  MoveL 4600 to (-46.03, -30.75, -4) mm, rotated rx 180 ry 0 rz 90 deg; joints [72.359, -18.311, 87.085, 0, 21.226, 72.359]
  Establecer velocidad (1000.0 mm/s)
  MoveL 4601 to (-46.03, -30.75, 10) mm, rotated rx -180 ry 0 rz 90 deg; joints [72.359, -19.035, 87.552, 0, 21.483, 72.359]
  Establecer velocidad (66.7 mm/s)
  MoveL 4602 to (16.92, -66.15, 10) mm, rotated rx -180 ry 0 rz 90 deg; joints [71.876, -17.66, 82.327, 0, 25.333, 71.876]
  MoveL 4603 to (16.92, -66.15, -3.75) mm, rotated rx 180 ry 0 rz 90 deg; joints [71.876, -16.964, 81.867, 0, 25.097, 71.876]
  MoveL 4604 to (16.76, -67.66, -4.16) mm, rotated rx 180 ry 0 rz 90 deg; joints [71.827, -16.937, 81.829, 0, 25.108, 71.827]
  MoveL 4605 to (16.96, -69.17, -4.56) mm, rotated rx -180 ry 0 rz 90 deg; joints [71.782, -16.903, 81.765, 0, 25.138, 71.782]
  MoveL 4606 to (17.5, -70.59, -4.97) mm, rotated rx 180 ry 0 rz 90 deg; joints [71.743, -16.862, 81.678, 0, 25.184, 71.743]
  MoveL 4607 to (18.34, -71.86, -5.37) mm, rotated rx -180 ry 0 rz 90 deg; joints [71.712, -16.816, 81.574, 0, 25.243, 71.712]
  MoveL 4608 to (19.43, -72.91, -5.78) mm, rotated rx -180 ry 0 rz 90 deg; joints [71.69, -16.767, 81.455, 0, 25.311, 71.69]
  MoveL 4609 to (20.74, -73.69, -6.19) mm, rotated rx 180 ry 0 rz 90 deg; joints [71.679, -16.714, 81.328, 0, 25.386, 71.679]
  MoveL 4610 to (22.18, -74.17, -6.59) mm, rotated rx 180 ry 0 rz 90 deg; joints [71.679, -16.662, 81.198, 0, 25.463, 71.679]
  MoveL 4611 to (23.69, -74.28, -7) mm, rotated rx 180 ry 0 rz 90 deg; joints [71.691, -16.609, 81.071, 0, 25.538, 71.691]
  MoveC 4612 to (36.25, -74.06, -7) mm, rotated rx 180 ry 0 rz 90 deg; joints [71.827, -16.352, 80.159, 0, 26.193, 71.827] to (48.8, -73.79, -7) mm, rotated rx -180 ry 0 rz 90 deg; joints [71.962, -16.087, 79.237, 0, 26.85, 71.962]
  MoveC 4613 to (51.44, -70.72, -7) mm, rotated rx -180 ry 0 rz 90 deg; joints [72.082, -16.052, 79.115, 0, 26.937, 72.082] to (51.58, -66.68, -7) mm, rotated rx 180 ry 0 rz 90 deg; joints [72.208, -16.077, 79.201, 0, 26.876, 72.208]
  MoveC 4614 to (38.79, -51.64, -7) mm, rotated rx 180 ry 0 rz 90 deg; joints [72.548, -16.449, 80.502, 0, 25.948, 72.548] to (25.93, -36.65, -7) mm, rotated rx -180 ry 0 rz 90 deg; joints [72.893, -16.807, 81.782, 0, 25.025, 72.893]
  MoveC 4615 to (25.5, -36.2, -7) mm, rotated rx 180 ry 0 rz 90 deg; joints [72.903, -16.818, 81.823, 0, 24.995, 72.903] to (25.04, -35.79, -7) mm, rotated rx -180 ry 0 rz 90 deg; joints [72.911, -16.83, 81.866, 0, 24.964, 72.911]
  MoveL 4616 to (12.33, -25.61, -7) mm, rotated rx 180 ry 0 rz 90 deg; joints [73.111, -17.14, 83.008, 0, 24.132, 73.111]
  MoveL 4617 to (11.85, -25.24, -7) mm, rotated rx -180 ry 0 rz 90 deg; joints [73.118, -17.151, 83.05, 0, 24.101, 73.118]
  MoveC 4618 to (9.1, -24.89, -7) mm, rotated rx 180 ry 0 rz 90 deg; joints [73.102, -17.206, 83.255, 0, 23.951, 73.102] to (6.64, -26.18, -7) mm, rotated rx -180 ry 0 rz 90 deg; joints [73.037, -17.245, 83.402, 0, 23.843, 73.037]
  MoveC 4619 to (6.25, -26.7, -7) mm, rotated rx 180 ry 0 rz 90 deg; joints [73.017, -17.25, 83.419, 0, 23.831, 73.017] to (6, -27.31, -7) mm, rotated rx 180 ry 0 rz 90 deg; joints [72.995, -17.251, 83.424, 0, 23.827, 72.995]
  MoveL 4620 to (-5.3, -69.65, -7) mm, rotated rx 180 ry 0 rz 90 deg; joints [71.534, -17.208, 83.264, 0, 23.945, 71.534]
  MoveC 4621 to (-4.6, -73.1, -7) mm, rotated rx 180 ry 0 rz 90 deg; joints [71.432, -17.173, 83.132, 0, 24.041, 71.432] to (-1.42, -74.62, -7) mm, rotated rx -180 ry 0 rz 90 deg; joints [71.418, -17.103, 82.87, 0, 24.233, 71.418]
  MoveC 4622 to (11.14, -74.47, -7) mm, rotated rx 180 ry 0 rz 90 deg; joints [71.555, -16.86, 81.975, 0, 24.885, 71.555] to (23.69, -74.28, -7) mm, rotated rx 180 ry 0 rz 90 deg; joints [71.691, -16.609, 81.071, 0, 25.538, 71.691]
  MoveL 4623 to (23.57, -66.73, -7) mm, rotated rx -180 ry 0 rz 90 deg; joints [71.925, -16.662, 81.261, 0, 25.401, 71.925]
  MoveL 4624 to (23.57, -66.73, -4) mm, rotated rx -180 ry 0 rz 90 deg; joints [71.925, -16.814, 81.363, 0, 25.451, 71.925]
  Establecer velocidad (1000.0 mm/s)
  MoveL 4625 to (23.57, -66.73, 10) mm, rotated rx 180 ry 0 rz 90 deg; joints [71.925, -17.521, 81.832, 0, 25.689, 71.925]
  Establecer velocidad (66.7 mm/s)
  MoveL 4626 to (64.23, -31.47, 10) mm, rotated rx -180 ry 0 rz 90 deg; joints [73.417, -16.891, 79.643, 0, 27.248, 73.417]
  MoveL 4627 to (64.23, -31.47, -3.75) mm, rotated rx 180 ry 0 rz 90 deg; joints [73.417, -16.202, 79.18, 0, 27.021, 73.417]
  MoveL 4628 to (65.74, -31.65, -4.16) mm, rotated rx 180 ry 0 rz 90 deg; joints [73.425, -16.147, 79.049, 0, 27.098, 73.425]
  MoveL 4629 to (67.24, -31.47, -4.56) mm, rotated rx -180 ry 0 rz 90 deg; joints [73.445, -16.095, 78.926, 0, 27.169, 73.445]
  MoveL 4630 to (68.68, -30.95, -4.97) mm, rotated rx -180 ry 0 rz 90 deg; joints [73.474, -16.046, 78.816, 0, 27.231, 73.474]
  MoveL 4631 to (69.96, -30.14, -5.37) mm, rotated rx 180 ry 0 rz 90 deg; joints [73.511, -16.003, 78.723, 0, 27.279, 73.511]
  MoveL 4632 to (71.03, -29.06, -5.78) mm, rotated rx 180 ry 0 rz 90 deg; joints [73.554, -15.966, 78.653, 0, 27.313, 73.554]
  MoveL 4633 to (71.83, -27.77, -6.19) mm, rotated rx 180 ry 0 rz 90 deg; joints [73.601, -15.936, 78.607, 0, 27.329, 73.601]
  MoveL 4634 to (72.33, -26.33, -6.59) mm, rotated rx -180 ry 0 rz 90 deg; joints [73.65, -15.914, 78.587, 0, 27.327, 73.65]
  MoveL 4635 to (72.47, -24.83, -7) mm, rotated rx 180 ry 0 rz 90 deg; joints [73.698, -15.9, 78.596, 0, 27.304, 73.698]
  MoveL 4636 to (72.47, -13.16, -7) mm, rotated rx 180 ry 0 rz 90 deg; joints [74.059, -15.975, 78.851, 0, 27.124, 74.059]
  MoveC 4637 to (70.6, -10.5, -7) mm, rotated rx 180 ry 0 rz 90 deg; joints [74.125, -16.033, 79.049, 0, 26.983, 74.125] to (67.76, -8.91, -7) mm, rotated rx 180 ry 0 rz 90 deg; joints [74.15, -16.105, 79.297, 0, 26.807, 74.15]
  MoveC 4638 to (66.52, -8.73, -7) mm, rotated rx 180 ry 0 rz 90 deg; joints [74.144, -16.133, 79.394, 0, 26.739, 74.144] to (65.29, -8.93, -7) mm, rotated rx 180 ry 0 rz 90 deg; joints [74.127, -16.158, 79.482, 0, 26.676, 74.127]
  MoveL 4639 to (65.23, -9, -7) mm, rotated rx 180 ry 0 rz 90 deg; joints [74.124, -16.159, 79.485, 0, 26.674, 74.124]
  MoveL 4640 to (54.8, -23.22, -7) mm, rotated rx 180 ry 0 rz 90 deg; joints [73.587, -16.295, 79.957, 0, 26.337, 73.587]
  MoveL 4641 to (54.33, -23.9, -7) mm, rotated rx -180 ry 0 rz 90 deg; joints [73.561, -16.3, 79.977, 0, 26.323, 73.561]
  MoveC 4642 to (53.72, -26.08, -7) mm, rotated rx -180 ry 0 rz 90 deg; joints [73.487, -16.299, 79.974, 0, 26.325, 73.487] to (54.54, -28.19, -7) mm, rotated rx -180 ry 0 rz 90 deg; joints [73.429, -16.269, 79.867, 0, 26.402, 73.429]
  MoveL 4643 to (55.12, -28.9, -7) mm, rotated rx 180 ry 0 rz 90 deg; joints [73.412, -16.252, 79.808, 0, 26.444, 73.412]
  MoveL 4644 to (65.68, -40.76, -7) mm, rotated rx 180 ry 0 rz 90 deg; joints [73.143, -15.946, 78.75, 0, 27.195, 73.143]
  MoveC 4645 to (68.07, -40.73, -7) mm, rotated rx 180 ry 0 rz 90 deg; joints [73.166, -15.893, 78.571, 0, 27.322, 73.166] to (70.2, -39.65, -7) mm, rotated rx 180 ry 0 rz 90 deg; joints [73.22, -15.853, 78.435, 0, 27.418, 73.22]
  MoveL 4646 to (70.46, -39.44, -7) mm, rotated rx 180 ry 0 rz 90 deg; joints [73.228, -15.849, 78.42, 0, 27.429, 73.228]
  MoveC 4647 to (71.67, -38.1, -7) mm, rotated rx -180 ry 0 rz 90 deg; joints [73.281, -15.831, 78.359, 0, 27.472, 73.281] to (72.47, -36.48, -7) mm, rotated rx -180 ry 0 rz 90 deg; joints [73.338, -15.824, 78.335, 0, 27.489, 73.338]
  MoveL 4648 to (72.47, -24.83, -7) mm, rotated rx 180 ry 0 rz 90 deg; joints [73.698, -15.9, 78.596, 0, 27.304, 73.698]
  MoveL 4649 to (64.92, -24.83, -7) mm, rotated rx -180 ry 0 rz 90 deg; joints [73.629, -16.066, 79.165, 0, 26.901, 73.629]
  MoveL 4650 to (64.92, -24.83, -4) mm, rotated rx 180 ry 0 rz 90 deg; joints [73.629, -16.217, 79.268, 0, 26.949, 73.629]
  Establecer velocidad (1000.0 mm/s)
  MoveL 4651 to (64.92, -24.83, 10) mm, rotated rx 180 ry 0 rz 90 deg; joints [73.629, -16.919, 79.739, 0, 27.18, 73.629]
  Establecer velocidad (66.7 mm/s)
  MoveL 4652 to (36.79, 21.66, 10) mm, rotated rx -180 ry 0 rz 90 deg; joints [74.843, -17.788, 82.79, 0, 24.998, 74.843]
  MoveL 4653 to (36.79, 21.66, -3.75) mm, rotated rx -180 ry 0 rz 90 deg; joints [74.843, -17.092, 82.33, 0, 24.762, 74.843]
  MoveL 4654 to (36.94, 23.17, -4.16) mm, rotated rx -180 ry 0 rz 90 deg; joints [74.892, -17.076, 82.335, 0, 24.741, 74.892]
  MoveL 4655 to (36.73, 24.67, -4.56) mm, rotated rx -180 ry 0 rz 90 deg; joints [74.939, -17.068, 82.366, 0, 24.702, 74.939]
  MoveL 4656 to (36.19, 26.09, -4.97) mm, rotated rx 180 ry 0 rz 90 deg; joints [74.979, -17.066, 82.42, 0, 24.646, 74.979]
  MoveL 4657 to (35.35, 27.36, -5.37) mm, rotated rx 180 ry 0 rz 90 deg; joints [75.013, -17.068, 82.492, 0, 24.576, 75.013]
  MoveL 4658 to (34.25, 28.4, -5.78) mm, rotated rx 180 ry 0 rz 90 deg; joints [75.037, -17.075, 82.579, 0, 24.496, 75.037]
  MoveL 4659 to (32.94, 29.18, -6.19) mm, rotated rx 180 ry 0 rz 90 deg; joints [75.05, -17.084, 82.675, 0, 24.409, 75.05]
  MoveL 4660 to (31.49, 29.65, -6.59) mm, rotated rx -180 ry 0 rz 90 deg; joints [75.053, -17.094, 82.776, 0, 24.319, 75.053]
  MoveL 4661 to (29.98, 29.76, -7) mm, rotated rx 180 ry 0 rz 90 deg; joints [75.043, -17.104, 82.874, 0, 24.23, 75.043]
  MoveL 4662 to (10.9, 29.36, -7) mm, rotated rx -180 ry 0 rz 90 deg; joints [74.865, -17.466, 84.239, 0, 23.226, 74.865]
  MoveL 4663 to (9.95, 29.33, -7) mm, rotated rx 180 ry 0 rz 90 deg; joints [74.856, -17.483, 84.306, 0, 23.177, 74.856]
  MoveC 4664 to (7.63, 28.6, -7) mm, rotated rx 180 ry 0 rz 90 deg; joints [74.812, -17.522, 84.457, 0, 23.065, 74.812] to (6.16, 26.68, -7) mm, rotated rx 180 ry 0 rz 90 deg; joints [74.736, -17.54, 84.525, 0, 23.015, 74.736]
  MoveC 4665 to (5.85, 25.43, -7) mm, rotated rx -180 ry 0 rz 90 deg; joints [74.693, -17.539, 84.523, 0, 23.016, 74.693] to (6.04, 24.17, -7) mm, rotated rx 180 ry 0 rz 90 deg; joints [74.653, -17.529, 84.485, 0, 23.045, 74.653]
  MoveL 4666 to (11.41, 9.41, -7) mm, rotated rx -180 ry 0 rz 90 deg; joints [74.225, -17.353, 83.809, 0, 23.544, 74.225]
  MoveC 4667 to (11.94, 8.41, -7) mm, rotated rx -180 ry 0 rz 90 deg; joints [74.197, -17.337, 83.75, 0, 23.587, 74.197] to (12.74, 7.59, -7) mm, rotated rx -180 ry 0 rz 90 deg; joints [74.178, -17.318, 83.676, 0, 23.642, 74.178]
  MoveL 4668 to (28.26, -4.36, -7) mm, rotated rx -180 ry 0 rz 90 deg; joints [73.937, -16.952, 82.311, 0, 24.64, 73.937]
  MoveC 4669 to (29.93, -5.1, -7) mm, rotated rx -180 ry 0 rz 90 deg; joints [73.929, -16.914, 82.175, 0, 24.74, 73.929] to (31.75, -4.99, -7) mm, rotated rx 180 ry 0 rz 90 deg; joints [73.949, -16.879, 82.045, 0, 24.834, 73.949]
  MoveC 4670 to (33.02, -4.44, -7) mm, rotated rx 180 ry 0 rz 90 deg; joints [73.978, -16.857, 81.963, 0, 24.893, 73.978] to (34.03, -3.48, -7) mm, rotated rx -180 ry 0 rz 90 deg; joints [74.018, -16.842, 81.91, 0, 24.932, 74.018]
  MoveL 4671 to (34.59, -2.74, -7) mm, rotated rx 180 ry 0 rz 90 deg; joints [74.047, -16.835, 81.885, 0, 24.95, 74.047]
  MoveL 4672 to (52.72, 22.78, -7) mm, rotated rx -180 ry 0 rz 90 deg; joints [75.015, -16.609, 81.071, 0, 25.538, 75.015]
  MoveC 4673 to (53.21, 23.87, -7) mm, rotated rx 180 ry 0 rz 90 deg; joints [75.054, -16.605, 81.056, 0, 25.549, 75.054] to (53.26, 25.07, -7) mm, rotated rx 180 ry 0 rz 90 deg; joints [75.092, -16.611, 81.076, 0, 25.534, 75.092]
  MoveL 4674 to (53.13, 25.86, -7) mm, rotated rx 180 ry 0 rz 90 deg; joints [75.116, -16.618, 81.101, 0, 25.516, 75.116]
  MoveC 4675 to (52.1, 28.37, -7) mm, rotated rx 180 ry 0 rz 90 deg; joints [75.187, -16.653, 81.227, 0, 25.426, 75.187] to (50.02, 30.11, -7) mm, rotated rx -180 ry 0 rz 90 deg; joints [75.225, -16.705, 81.415, 0, 25.29, 75.225]
  MoveL 4676 to (45.96, 30.09, -7) mm, rotated rx -180 ry 0 rz 90 deg; joints [75.19, -16.788, 81.713, 0, 25.075, 75.19]
  MoveL 4677 to (29.98, 29.76, -7) mm, rotated rx 180 ry 0 rz 90 deg; joints [75.043, -17.104, 82.874, 0, 24.23, 75.043]
  MoveL 4678 to (30.14, 22.21, -7) mm, rotated rx 180 ry 0 rz 90 deg; joints [74.803, -17.061, 82.715, 0, 24.346, 74.803]
  MoveL 4679 to (30.14, 22.21, -4) mm, rotated rx 180 ry 0 rz 90 deg; joints [74.803, -17.214, 82.816, 0, 24.397, 74.803]
  Establecer velocidad (1000.0 mm/s)
  MoveL 4680 to (30.14, 22.21, 10) mm, rotated rx 180 ry 0 rz 90 deg; joints [74.803, -17.924, 83.285, 0, 24.64, 74.803]
  Establecer velocidad (66.7 mm/s)
  MoveL 4681 to (27.33, 65.77, 10) mm, rotated rx -180 ry 0 rz 90 deg; joints [76.185, -18.2, 84.303, 0, 23.897, 76.185]
  MoveL 4682 to (27.33, 65.77, -3.75) mm, rotated rx -180 ry 0 rz 90 deg; joints [76.185, -17.499, 83.844, 0, 23.655, 76.185]
  MoveL 4683 to (27.54, 67.27, -4.16) mm, rotated rx 180 ry 0 rz 90 deg; joints [76.236, -17.481, 83.842, 0, 23.64, 76.236]
  MoveL 4684 to (27.39, 68.78, -4.56) mm, rotated rx 180 ry 0 rz 90 deg; joints [76.284, -17.471, 83.866, 0, 23.605, 76.284]
  MoveL 4685 to (26.9, 70.22, -4.97) mm, rotated rx -180 ry 0 rz 90 deg; joints [76.327, -17.466, 83.913, 0, 23.553, 76.327]
  MoveL 4686 to (26.11, 71.51, -5.37) mm, rotated rx 180 ry 0 rz 90 deg; joints [76.363, -17.466, 83.979, 0, 23.487, 76.363]
  MoveL 4687 to (25.04, 72.6, -5.78) mm, rotated rx 180 ry 0 rz 90 deg; joints [76.39, -17.47, 84.061, 0, 23.41, 76.39]
  MoveL 4688 to (23.77, 73.43, -6.19) mm, rotated rx 180 ry 0 rz 90 deg; joints [76.407, -17.477, 84.153, 0, 23.324, 76.407]
  MoveL 4689 to (22.34, 73.95, -6.59) mm, rotated rx 180 ry 0 rz 90 deg; joints [76.413, -17.486, 84.251, 0, 23.235, 76.413]
  MoveL 4690 to (20.84, 74.12, -7) mm, rotated rx 180 ry 0 rz 90 deg; joints [76.406, -17.494, 84.348, 0, 23.146, 76.406]
  MoveL 4691 to (12.79, 74.25, -7) mm, rotated rx 180 ry 0 rz 90 deg; joints [76.347, -17.643, 84.926, 0, 22.717, 76.347]
  MoveL 4692 to (-26.06, 74.73, -7) mm, rotated rx 180 ry 0 rz 90 deg; joints [76.046, -18.319, 87.663, 0, 20.656, 76.046]
  MoveL 4693 to (-27.17, 74.74, -7) mm, rotated rx -180 ry 0 rz 90 deg; joints [76.037, -18.338, 87.74, 0, 20.597, 76.037]
  MoveC 4694 to (-29.75, 71.47, -7) mm, rotated rx 180 ry 0 rz 90 deg; joints [75.905, -18.366, 87.862, 0, 20.504, 75.905] to (-29.32, 67.32, -7) mm, rotated rx 180 ry 0 rz 90 deg; joints [75.77, -18.342, 87.76, 0, 20.582, 75.77]
  MoveL 4695 to (-10.07, 55.09, -7) mm, rotated rx 180 ry 0 rz 90 deg; joints [75.526, -17.965, 86.203, 0, 21.762, 75.526]
  MoveC 4696 to (-8.73, 54.52, -7) mm, rotated rx 180 ry 0 rz 90 deg; joints [75.519, -17.939, 86.099, 0, 21.84, 75.519] to (-7.29, 54.39, -7) mm, rotated rx 180 ry 0 rz 90 deg; joints [75.527, -17.913, 85.996, 0, 21.918, 75.527]
  MoveL 4697 to (-6.16, 54.47, -7) mm, rotated rx -180 ry 0 rz 90 deg; joints [75.539, -17.894, 85.918, 0, 21.976, 75.539]
  MoveL 4698 to (27.01, 56.93, -7) mm, rotated rx 180 ry 0 rz 90 deg; joints [75.896, -17.297, 83.599, 0, 23.699, 75.896]
  MoveL 4699 to (33.64, 57.46, -7) mm, rotated rx -180 ry 0 rz 90 deg; joints [75.967, -17.172, 83.128, 0, 24.044, 75.967]
  MoveC 4700 to (51.29, 59.11, -7) mm, rotated rx -180 ry 0 rz 90 deg; joints [76.161, -16.83, 81.867, 0, 24.963, 76.161] to (68.87, 61.29, -7) mm, rotated rx 180 ry 0 rz 90 deg; joints [76.367, -16.477, 80.6, 0, 25.877, 76.367]
  MoveC 4701 to (70.75, 62.3, -7) mm, rotated rx 180 ry 0 rz 90 deg; joints [76.414, -16.442, 80.478, 0, 25.965, 76.414] to (71.5, 64.29, -7) mm, rotated rx -180 ry 0 rz 90 deg; joints [76.483, -16.437, 80.458, 0, 25.979, 76.483]
  MoveL 4702 to (71.51, 68.7, -7) mm, rotated rx 180 ry 0 rz 90 deg; joints [76.623, -16.459, 80.536, 0, 25.923, 76.623]
  MoveL 4703 to (71.5, 69.4, -7) mm, rotated rx 180 ry 0 rz 90 deg; joints [76.645, -16.463, 80.549, 0, 25.914, 76.645]
  MoveC 4704 to (70.71, 71.35, -7) mm, rotated rx 180 ry 0 rz 90 deg; joints [76.702, -16.489, 80.643, 0, 25.846, 76.702] to (68.8, 72.25, -7) mm, rotated rx -180 ry 0 rz 90 deg; joints [76.716, -16.534, 80.801, 0, 25.732, 76.716]
  MoveC 4705 to (45.55, 73.46, -7) mm, rotated rx 180 ry 0 rz 90 deg; joints [76.577, -17.015, 82.544, 0, 24.471, 76.577] to (22.27, 74.09, -7) mm, rotated rx -180 ry 0 rz 90 deg; joints [76.417, -17.467, 84.245, 0, 23.222, 76.417]
  MoveL 4706 to (20.84, 74.12, -7) mm, rotated rx 180 ry 0 rz 90 deg; joints [76.406, -17.494, 84.348, 0, 23.146, 76.406]
  MoveL 4707 to (20.71, 66.57, -7) mm, rotated rx 180 ry 0 rz 90 deg; joints [76.158, -17.462, 84.225, 0, 23.237, 76.158]
  MoveL 4708 to (20.71, 66.57, -4) mm, rotated rx 180 ry 0 rz 90 deg; joints [76.158, -17.615, 84.327, 0, 23.288, 76.158]
  Establecer velocidad (1000.0 mm/s)
  MoveL 4709 to (20.71, 66.57, 10) mm, rotated rx 180 ry 0 rz 90 deg; joints [76.158, -18.33, 84.794, 0, 23.536, 76.158]
  Establecer velocidad (66.7 mm/s)
  MoveL 4710 to (27.32, 65.52, 10) mm, rotated rx 180 ry 0 rz 90 deg; joints [76.177, -18.199, 84.299, 0, 23.899, 76.177]
  MoveL 4711 to (27.32, 65.52, -4) mm, rotated rx 180 ry 0 rz 90 deg; joints [76.177, -17.485, 83.832, 0, 23.653, 76.177]
  MoveL 4712 to (27.53, 67.02, -4.41) mm, rotated rx 180 ry 0 rz 90 deg; joints [76.228, -17.468, 83.83, 0, 23.638, 76.228]
  MoveL 4713 to (27.38, 68.53, -4.81) mm, rotated rx -180 ry 0 rz 90 deg; joints [76.276, -17.457, 83.854, 0, 23.603, 76.276]
  MoveL 4714 to (26.89, 69.97, -5.22) mm, rotated rx 180 ry 0 rz 90 deg; joints [76.319, -17.452, 83.9, 0, 23.552, 76.319]
  MoveL 4715 to (26.1, 71.27, -5.63) mm, rotated rx 180 ry 0 rz 90 deg; joints [76.355, -17.452, 83.966, 0, 23.486, 76.355]
  MoveL 4716 to (25.04, 72.36, -6.03) mm, rotated rx -180 ry 0 rz 90 deg; joints [76.382, -17.457, 84.048, 0, 23.408, 76.382]
  MoveL 4717 to (23.76, 73.19, -6.44) mm, rotated rx 180 ry 0 rz 90 deg; joints [76.399, -17.464, 84.141, 0, 23.323, 76.399]
  MoveL 4718 to (22.34, 73.71, -6.84) mm, rotated rx 180 ry 0 rz 90 deg; joints [76.405, -17.472, 84.239, 0, 23.234, 76.405]
  MoveL 4719 to (20.83, 73.88, -7.25) mm, rotated rx -180 ry 0 rz 90 deg; joints [76.398, -17.48, 84.336, 0, 23.144, 76.398]
  MoveC 4720 to (-2.85, 74.25, -7.25) mm, rotated rx 180 ry 0 rz 90 deg; joints [76.221, -17.91, 86.027, 0, 21.884, 76.221] to (-26.54, 74.55, -7.25) mm, rotated rx -180 ry 0 rz 90 deg; joints [76.035, -18.314, 87.685, 0, 20.629, 76.035]
  MoveC 4721 to (-29.11, 71.31, -7.25) mm, rotated rx -180 ry 0 rz 90 deg; joints [75.905, -18.342, 87.806, 0, 20.536, 75.905] to (-28.68, 67.2, -7.25) mm, rotated rx -180 ry 0 rz 90 deg; joints [75.771, -18.318, 87.706, 0, 20.613, 75.771]
  MoveL 4722 to (-27.01, 66.12, -7.25) mm, rotated rx -180 ry 0 rz 90 deg; joints [75.749, -18.286, 87.571, 0, 20.716, 75.749]
  MoveL 4723 to (-11.7, 56.39, -7.25) mm, rotated rx 180 ry 0 rz 90 deg; joints [75.555, -17.986, 86.332, 0, 21.654, 75.555]
  MoveL 4724 to (-9.95, 55.27, -7.25) mm, rotated rx -180 ry 0 rz 90 deg; joints [75.533, -17.951, 86.19, 0, 21.761, 75.533]
  MoveC 4725 to (-8.59, 54.68, -7.25) mm, rotated rx 180 ry 0 rz 90 deg; joints [75.526, -17.925, 86.084, 0, 21.841, 75.526] to (-7.11, 54.59, -7.25) mm, rotated rx 180 ry 0 rz 90 deg; joints [75.535, -17.898, 85.978, 0, 21.92, 75.535]
  MoveL 4726 to (-6.16, 54.66, -7.25) mm, rotated rx 180 ry 0 rz 90 deg; joints [75.545, -17.882, 85.913, 0, 21.969, 75.545]
  MoveL 4727 to (25.11, 56.98, -7.25) mm, rotated rx 180 ry 0 rz 90 deg; joints [75.882, -17.321, 83.728, 0, 23.593, 75.882]
  MoveL 4728 to (32.69, 57.59, -7.25) mm, rotated rx 180 ry 0 rz 90 deg; joints [75.964, -17.178, 83.191, 0, 23.988, 75.964]
  MoveC 4729 to (50.72, 59.32, -7.25) mm, rotated rx 180 ry 0 rz 90 deg; joints [76.163, -16.83, 81.904, 0, 24.926, 76.163] to (68.69, 61.63, -7.25) mm, rotated rx 180 ry 0 rz 90 deg; joints [76.377, -16.47, 80.611, 0, 25.859, 76.377]
  MoveC 4730 to (70.41, 62.54, -7.25) mm, rotated rx 180 ry 0 rz 90 deg; joints [76.419, -16.438, 80.499, 0, 25.939, 76.419] to (71.16, 64.33, -7.25) mm, rotated rx 180 ry 0 rz 90 deg; joints [76.482, -16.432, 80.475, 0, 25.957, 76.482]
  MoveC 4731 to (71.23, 66.85, -7.25) mm, rotated rx -180 ry 0 rz 90 deg; joints [76.562, -16.443, 80.515, 0, 25.928, 76.562] to (71.16, 69.37, -7.25) mm, rotated rx -180 ry 0 rz 90 deg; joints [76.642, -16.457, 80.566, 0, 25.891, 76.642]
  MoveC 4732 to (70.37, 71.13, -7.25) mm, rotated rx -180 ry 0 rz 90 deg; joints [76.692, -16.483, 80.656, 0, 25.827, 76.692] to (68.62, 71.93, -7.25) mm, rotated rx 180 ry 0 rz 90 deg; joints [76.704, -16.523, 80.801, 0, 25.723, 76.704]
  MoveC 4733 to (46.88, 73.13, -7.25) mm, rotated rx 180 ry 0 rz 90 deg; joints [76.577, -16.974, 82.432, 0, 24.542, 76.577] to (25.11, 73.8, -7.25) mm, rotated rx 180 ry 0 rz 90 deg; joints [76.429, -17.4, 84.027, 0, 23.373, 76.429]
  MoveC 4734 to (22.97, 73.84, -7.25) mm, rotated rx -180 ry 0 rz 90 deg; joints [76.414, -17.44, 84.182, 0, 23.258, 76.414] to (20.83, 73.88, -7.25) mm, rotated rx 180 ry 0 rz 90 deg; joints [76.398, -17.48, 84.336, 0, 23.144, 76.398]
  MoveL 4735 to (20.7, 66.33, -7.25) mm, rotated rx -180 ry 0 rz 90 deg; joints [76.15, -17.448, 84.213, 0, 23.235, 76.15]
  MoveL 4736 to (20.7, 66.33, -4.25) mm, rotated rx -180 ry 0 rz 90 deg; joints [76.15, -17.602, 84.315, 0, 23.287, 76.15]
  Establecer velocidad (1000.0 mm/s)
  MoveL 4737 to (20.7, 66.33, 10) mm, rotated rx -180 ry 0 rz 90 deg; joints [76.15, -18.329, 84.791, 0, 23.539, 76.15]
  Establecer velocidad (66.7 mm/s)
  MoveL 4738 to (36.06, 21.39, 10) mm, rotated rx -180 ry 0 rz 90 deg; joints [74.828, -17.802, 82.838, 0, 24.964, 74.828]
  MoveL 4739 to (36.06, 21.39, -4) mm, rotated rx 180 ry 0 rz 90 deg; joints [74.828, -17.092, 82.37, 0, 24.723, 74.828]
  MoveL 4740 to (36.22, 22.9, -4.41) mm, rotated rx -180 ry 0 rz 90 deg; joints [74.878, -17.076, 82.374, 0, 24.702, 74.878]
  MoveL 4741 to (36, 24.41, -4.81) mm, rotated rx -180 ry 0 rz 90 deg; joints [74.924, -17.068, 82.405, 0, 24.663, 74.924]
  MoveL 4742 to (35.46, 25.83, -5.22) mm, rotated rx 180 ry 0 rz 90 deg; joints [74.965, -17.066, 82.459, 0, 24.607, 74.965]
  MoveL 4743 to (34.62, 27.09, -5.63) mm, rotated rx -180 ry 0 rz 90 deg; joints [74.998, -17.069, 82.531, 0, 24.537, 74.998]
  MoveL 4744 to (33.52, 28.14, -6.03) mm, rotated rx 180 ry 0 rz 90 deg; joints [75.022, -17.075, 82.618, 0, 24.457, 75.022]
  MoveL 4745 to (32.22, 28.92, -6.44) mm, rotated rx -180 ry 0 rz 90 deg; joints [75.036, -17.084, 82.714, 0, 24.37, 75.036]
  MoveL 4746 to (30.77, 29.39, -6.84) mm, rotated rx -180 ry 0 rz 90 deg; joints [75.039, -17.095, 82.814, 0, 24.28, 75.039]
  MoveL 4747 to (29.26, 29.5, -7.25) mm, rotated rx -180 ry 0 rz 90 deg; joints [75.029, -17.104, 82.913, 0, 24.191, 75.029]
  MoveL 4748 to (13.74, 29.19, -7.25) mm, rotated rx 180 ry 0 rz 90 deg; joints [74.885, -17.399, 84.024, 0, 23.375, 74.885]
  MoveL 4749 to (9.95, 29.11, -7.25) mm, rotated rx 180 ry 0 rz 90 deg; joints [74.849, -17.469, 84.294, 0, 23.176, 74.849]
  MoveL 4750 to (9, 28.95, -7.25) mm, rotated rx -180 ry 0 rz 90 deg; joints [74.835, -17.486, 84.358, 0, 23.128, 74.835]
  MoveC 4751 to (6.86, 27.27, -7.25) mm, rotated rx -180 ry 0 rz 90 deg; joints [74.762, -17.517, 84.478, 0, 23.039, 74.762] to (6.17, 24.64, -7.25) mm, rotated rx 180 ry 0 rz 90 deg; joints [74.67, -17.517, 84.476, 0, 23.041, 74.67]
  MoveL 4752 to (6.29, 24.17, -7.25) mm, rotated rx -180 ry 0 rz 90 deg; joints [74.656, -17.512, 84.458, 0, 23.054, 74.656]
  MoveL 4753 to (6.64, 23.22, -7.25) mm, rotated rx -180 ry 0 rz 90 deg; joints [74.628, -17.501, 84.415, 0, 23.086, 74.628]
  MoveL 4754 to (11.66, 9.42, -7.25) mm, rotated rx 180 ry 0 rz 90 deg; joints [74.227, -17.335, 83.782, 0, 23.553, 74.227]
  MoveC 4755 to (12.05, 8.66, -7.25) mm, rotated rx 180 ry 0 rz 90 deg; joints [74.206, -17.324, 83.739, 0, 23.585, 74.206] to (12.61, 8.02, -7.25) mm, rotated rx -180 ry 0 rz 90 deg; joints [74.191, -17.31, 83.686, 0, 23.624, 74.191]
  MoveL 4756 to (12.79, 7.85, -7.25) mm, rotated rx -180 ry 0 rz 90 deg; joints [74.187, -17.306, 83.669, 0, 23.636, 74.187]
  MoveL 4757 to (27.96, -3.81, -7.25) mm, rotated rx 180 ry 0 rz 90 deg; joints [73.952, -16.948, 82.337, 0, 24.612, 73.952]
  MoveL 4758 to (28.9, -4.48, -7.25) mm, rotated rx 180 ry 0 rz 90 deg; joints [73.94, -16.926, 82.254, 0, 24.672, 73.94]
  MoveC 4759 to (31.69, -4.67, -7.25) mm, rotated rx -180 ry 0 rz 90 deg; joints [73.959, -16.869, 82.047, 0, 24.822, 73.959] to (34.01, -3.1, -7.25) mm, rotated rx 180 ry 0 rz 90 deg; joints [74.03, -16.832, 81.911, 0, 24.921, 74.03]
  MoveL 4760 to (34.56, -2.37, -7.25) mm, rotated rx -180 ry 0 rz 90 deg; joints [74.058, -16.825, 81.886, 0, 24.939, 74.058]
  MoveL 4761 to (52.59, 23.08, -7.25) mm, rotated rx -180 ry 0 rz 90 deg; joints [75.023, -16.601, 81.078, 0, 25.523, 75.023]
  MoveC 4762 to (52.24, 27, -7.25) mm, rotated rx 180 ry 0 rz 90 deg; joints [75.145, -16.63, 81.181, 0, 25.449, 75.145] to (49.53, 29.85, -7.25) mm, rotated rx -180 ry 0 rz 90 deg; joints [75.212, -16.701, 81.437, 0, 25.264, 75.212]
  MoveL 4763 to (45.96, 29.83, -7.25) mm, rotated rx 180 ry 0 rz 90 deg; joints [75.182, -16.774, 81.7, 0, 25.074, 75.182]
  MoveL 4764 to (29.26, 29.5, -7.25) mm, rotated rx -180 ry 0 rz 90 deg; joints [75.029, -17.104, 82.913, 0, 24.191, 75.029]
  MoveL 4765 to (29.41, 21.95, -7.25) mm, rotated rx 180 ry 0 rz 90 deg; joints [74.788, -17.061, 82.754, 0, 24.307, 74.788]
  MoveL 4766 to (29.41, 21.95, -4.25) mm, rotated rx -180 ry 0 rz 90 deg; joints [74.788, -17.214, 82.856, 0, 24.358, 74.788]
  Establecer velocidad (1000.0 mm/s)
  MoveL 4767 to (29.41, 21.95, 10) mm, rotated rx 180 ry 0 rz 90 deg; joints [74.788, -17.937, 83.332, 0, 24.605, 74.788]
  Establecer velocidad (66.7 mm/s)
  MoveL 4768 to (63.96, -31.55, 10) mm, rotated rx -180 ry 0 rz 90 deg; joints [73.412, -16.896, 79.662, 0, 27.235, 73.412]
  MoveL 4769 to (63.96, -31.55, -4) mm, rotated rx 180 ry 0 rz 90 deg; joints [73.412, -16.195, 79.19, 0, 27.004, 73.412]
  MoveL 4770 to (65.46, -31.73, -4.41) mm, rotated rx -180 ry 0 rz 90 deg; joints [73.42, -16.14, 79.059, 0, 27.081, 73.42]
  MoveL 4771 to (66.97, -31.55, -4.81) mm, rotated rx 180 ry 0 rz 90 deg; joints [73.44, -16.088, 78.936, 0, 27.152, 73.44]
  MoveL 4772 to (68.4, -31.04, -5.22) mm, rotated rx 180 ry 0 rz 90 deg; joints [73.469, -16.039, 78.826, 0, 27.213, 73.469]
  MoveL 4773 to (69.68, -30.22, -5.63) mm, rotated rx 180 ry 0 rz 90 deg; joints [73.506, -15.996, 78.734, 0, 27.262, 73.506]
  MoveL 4774 to (70.76, -29.14, -6.03) mm, rotated rx -180 ry 0 rz 90 deg; joints [73.549, -15.959, 78.663, 0, 27.296, 73.549]
  MoveL 4775 to (71.56, -27.85, -6.44) mm, rotated rx -180 ry 0 rz 90 deg; joints [73.596, -15.929, 78.617, 0, 27.312, 73.596]
  MoveL 4776 to (72.06, -26.42, -6.84) mm, rotated rx 180 ry 0 rz 90 deg; joints [73.645, -15.907, 78.597, 0, 27.31, 73.645]
  MoveL 4777 to (72.2, -24.91, -7.25) mm, rotated rx -180 ry 0 rz 90 deg; joints [73.693, -15.893, 78.606, 0, 27.287, 73.693]
  MoveL 4778 to (72.2, -13.88, -7.25) mm, rotated rx 180 ry 0 rz 90 deg; joints [74.035, -15.964, 78.847, 0, 27.117, 74.035]
  MoveC 4779 to (70.43, -11.3, -7.25) mm, rotated rx -180 ry 0 rz 90 deg; joints [74.099, -16.019, 79.036, 0, 26.983, 74.099] to (67.76, -9.69, -7.25) mm, rotated rx 180 ry 0 rz 90 deg; joints [74.125, -16.087, 79.272, 0, 26.815, 74.125]
  MoveC 4780 to (66.44, -9.46, -7.25) mm, rotated rx 180 ry 0 rz 90 deg; joints [74.121, -16.117, 79.376, 0, 26.741, 74.121] to (65.12, -9.62, -7.25) mm, rotated rx 180 ry 0 rz 90 deg; joints [74.104, -16.145, 79.472, 0, 26.673, 74.104]
  MoveL 4781 to (55.13, -23.22, -7.25) mm, rotated rx 180 ry 0 rz 90 deg; joints [73.59, -16.275, 79.924, 0, 26.351, 73.59]
  MoveL 4782 to (54.65, -23.93, -7.25) mm, rotated rx 180 ry 0 rz 90 deg; joints [73.563, -16.281, 79.944, 0, 26.336, 73.563]
  MoveC 4783 to (54.05, -26.08, -7.25) mm, rotated rx -180 ry 0 rz 90 deg; joints [73.49, -16.28, 79.942, 0, 26.338, 73.49] to (54.86, -28.16, -7.25) mm, rotated rx 180 ry 0 rz 90 deg; joints [73.433, -16.249, 79.835, 0, 26.414, 73.433]
  MoveL 4784 to (55.44, -28.85, -7.25) mm, rotated rx 180 ry 0 rz 90 deg; joints [73.417, -16.233, 79.777, 0, 26.456, 73.417]
  MoveL 4785 to (65.51, -40.15, -7.25) mm, rotated rx 180 ry 0 rz 90 deg; joints [73.16, -15.941, 78.769, 0, 27.172, 73.16]
  MoveC 4786 to (68.03, -40.02, -7.25) mm, rotated rx 180 ry 0 rz 90 deg; joints [73.188, -15.886, 78.582, 0, 27.305, 73.188] to (70.24, -38.8, -7.25) mm, rotated rx 180 ry 0 rz 90 deg; joints [73.246, -15.845, 78.443, 0, 27.403, 73.246]
  MoveC 4787 to (71.39, -37.49, -7.25) mm, rotated rx 180 ry 0 rz 90 deg; joints [73.297, -15.829, 78.385, 0, 27.443, 73.297] to (72.2, -35.94, -7.25) mm, rotated rx 180 ry 0 rz 90 deg; joints [73.352, -15.821, 78.359, 0, 27.462, 73.352]
  MoveL 4788 to (72.2, -24.91, -7.25) mm, rotated rx -180 ry 0 rz 90 deg; joints [73.693, -15.893, 78.606, 0, 27.287, 73.693]
  MoveL 4789 to (64.65, -24.91, -7.25) mm, rotated rx -180 ry 0 rz 90 deg; joints [73.624, -16.059, 79.175, 0, 26.884, 73.624]
  MoveL 4790 to (64.65, -24.91, -4.25) mm, rotated rx 180 ry 0 rz 90 deg; joints [73.624, -16.21, 79.278, 0, 26.932, 73.624]
  Establecer velocidad (1000.0 mm/s)
  MoveL 4791 to (64.65, -24.91, 10) mm, rotated rx 180 ry 0 rz 90 deg; joints [73.624, -16.924, 79.757, 0, 27.167, 73.624]
  Establecer velocidad (66.7 mm/s)
  MoveL 4792 to (16.48, -65.93, 10) mm, rotated rx 180 ry 0 rz 90 deg; joints [71.878, -17.67, 82.364, 0, 25.306, 71.878]
  MoveL 4793 to (16.48, -65.93, -4) mm, rotated rx -180 ry 0 rz 90 deg; joints [71.878, -16.962, 81.895, 0, 25.067, 71.878]
  MoveL 4794 to (16.32, -67.44, -4.41) mm, rotated rx 180 ry 0 rz 90 deg; joints [71.829, -16.935, 81.857, 0, 25.077, 71.829]
  MoveL 4795 to (16.53, -68.94, -4.81) mm, rotated rx 180 ry 0 rz 90 deg; joints [71.784, -16.9, 81.793, 0, 25.107, 71.784]
  MoveL 4796 to (17.06, -70.37, -5.22) mm, rotated rx -180 ry 0 rz 90 deg; joints [71.745, -16.859, 81.707, 0, 25.153, 71.745]
  MoveL 4797 to (17.9, -71.63, -5.63) mm, rotated rx 180 ry 0 rz 90 deg; joints [71.714, -16.814, 81.602, 0, 25.212, 71.714]
  MoveL 4798 to (19, -72.68, -6.03) mm, rotated rx -180 ry 0 rz 90 deg; joints [71.693, -16.764, 81.483, 0, 25.281, 71.693]
  MoveL 4799 to (20.3, -73.47, -6.44) mm, rotated rx 180 ry 0 rz 90 deg; joints [71.682, -16.712, 81.357, 0, 25.356, 71.682]
  MoveL 4800 to (21.75, -73.94, -6.84) mm, rotated rx -180 ry 0 rz 90 deg; joints [71.682, -16.659, 81.226, 0, 25.433, 71.682]
  MoveL 4801 to (23.26, -74.06, -7.25) mm, rotated rx -180 ry 0 rz 90 deg; joints [71.694, -16.607, 81.1, 0, 25.507, 71.694]
  MoveC 4802 to (35.8, -73.82, -7.25) mm, rotated rx -180 ry 0 rz 90 deg; joints [71.83, -16.35, 80.189, 0, 26.161, 71.83] to (48.33, -73.53, -7.25) mm, rotated rx 180 ry 0 rz 90 deg; joints [71.965, -16.087, 79.269, 0, 26.817, 71.965]
  MoveC 4803 to (50.92, -70.47, -7.25) mm, rotated rx -180 ry 0 rz 90 deg; joints [72.085, -16.052, 79.151, 0, 26.902, 72.085] to (51.06, -66.46, -7.25) mm, rotated rx 180 ry 0 rz 90 deg; joints [72.21, -16.077, 79.236, 0, 26.841, 72.21]
  MoveC 4804 to (38.31, -51.44, -7.25) mm, rotated rx 180 ry 0 rz 90 deg; joints [72.55, -16.448, 80.533, 0, 25.915, 72.55] to (25.48, -36.48, -7.25) mm, rotated rx 180 ry 0 rz 90 deg; joints [72.894, -16.804, 81.81, 0, 24.994, 72.894]
  MoveL 4805 to (25.11, -36.14, -7.25) mm, rotated rx 180 ry 0 rz 90 deg; joints [72.901, -16.814, 81.844, 0, 24.969, 72.901]
  MoveL 4806 to (20.82, -32.69, -7.25) mm, rotated rx 180 ry 0 rz 90 deg; joints [72.968, -16.92, 82.232, 0, 24.688, 72.968]
  MoveL 4807 to (19.65, -31.75, -7.25) mm, rotated rx 180 ry 0 rz 90 deg; joints [72.987, -16.948, 82.337, 0, 24.611, 72.987]
  MoveL 4808 to (12.56, -26.06, -7.25) mm, rotated rx -180 ry 0 rz 90 deg; joints [73.099, -17.12, 82.973, 0, 24.148, 73.099]
  MoveL 4809 to (12.22, -25.78, -7.25) mm, rotated rx -180 ry 0 rz 90 deg; joints [73.104, -17.128, 83.003, 0, 24.125, 73.104]
  MoveC 4810 to (9.73, -25.16, -7.25) mm, rotated rx 180 ry 0 rz 90 deg; joints [73.1, -17.18, 83.195, 0, 23.984, 73.1] to (7.32, -26.06, -7.25) mm, rotated rx -180 ry 0 rz 90 deg; joints [73.048, -17.22, 83.348, 0, 23.873, 73.048]
  MoveL 4811 to (7.22, -26.13, -7.25) mm, rotated rx 180 ry 0 rz 90 deg; joints [73.045, -17.222, 83.353, 0, 23.868, 73.045]
  MoveC 4812 to (6.54, -26.82, -7.25) mm, rotated rx 180 ry 0 rz 90 deg; joints [73.016, -17.231, 83.387, 0, 23.844, 73.016] to (6.13, -27.7, -7.25) mm, rotated rx 180 ry 0 rz 90 deg; joints [72.984, -17.233, 83.397, 0, 23.836, 72.984]
  MoveL 4813 to (-5.06, -69.65, -7.25) mm, rotated rx 180 ry 0 rz 90 deg; joints [71.537, -17.191, 83.239, 0, 23.953, 71.537]
  MoveC 4814 to (-5.09, -71.39, -7.25) mm, rotated rx 180 ry 0 rz 90 deg; joints [71.481, -17.181, 83.199, 0, 23.982, 71.481] to (-4.26, -72.93, -7.25) mm, rotated rx -180 ry 0 rz 90 deg; joints [71.441, -17.155, 83.104, 0, 24.051, 71.441]
  MoveC 4815 to (-3.18, -73.89, -7.25) mm, rotated rx -180 ry 0 rz 90 deg; joints [71.423, -17.129, 83.004, 0, 24.125, 71.423] to (-1.82, -74.39, -7.25) mm, rotated rx 180 ry 0 rz 90 deg; joints [71.421, -17.099, 82.895, 0, 24.204, 71.421]
  MoveC 4816 to (10.72, -74.25, -7.25) mm, rotated rx 180 ry 0 rz 90 deg; joints [71.558, -16.857, 82.002, 0, 24.855, 71.558] to (23.26, -74.06, -7.25) mm, rotated rx -180 ry 0 rz 90 deg; joints [71.694, -16.607, 81.1, 0, 25.507, 71.694]
  MoveL 4817 to (23.13, -66.51, -7.25) mm, rotated rx -180 ry 0 rz 90 deg; joints [71.928, -16.66, 81.29, 0, 25.37, 71.928]
  MoveL 4818 to (23.13, -66.51, -4.25) mm, rotated rx -180 ry 0 rz 90 deg; joints [71.928, -16.812, 81.392, 0, 25.42, 71.928]
  Establecer velocidad (1000.0 mm/s)
  MoveL 4819 to (23.13, -66.51, 10) mm, rotated rx 180 ry 0 rz 90 deg; joints [71.928, -17.531, 81.869, 0, 25.662, 71.928]
  Establecer velocidad (66.7 mm/s)
  MoveL 4820 to (-35.06, -51.48, 10) mm, rotated rx 180 ry 0 rz 90 deg; joints [71.8, -18.73, 86.336, 0, 22.394, 71.8]
  MoveL 4821 to (-35.06, -51.48, -4) mm, rotated rx 180 ry 0 rz 90 deg; joints [71.8, -18.011, 85.869, 0, 22.141, 71.8]
  MoveL 4822 to (-33.65, -52.04, -4.41) mm, rotated rx -180 ry 0 rz 90 deg; joints [71.797, -17.962, 85.745, 0, 22.217, 71.797]
  MoveL 4823 to (-32.14, -52.25, -4.81) mm, rotated rx -180 ry 0 rz 90 deg; joints [71.806, -17.914, 85.623, 0, 22.291, 71.806]
  MoveL 4824 to (-30.63, -52.11, -5.22) mm, rotated rx -180 ry 0 rz 90 deg; joints [71.826, -17.867, 85.507, 0, 22.36, 71.826]
  MoveL 4825 to (-29.18, -51.65, -5.63) mm, rotated rx 180 ry 0 rz 90 deg; joints [71.857, -17.824, 85.404, 0, 22.42, 71.857]
  MoveL 4826 to (-27.87, -50.87, -6.03) mm, rotated rx 180 ry 0 rz 90 deg; joints [71.895, -17.784, 85.317, 0, 22.467, 71.895]
  MoveL 4827 to (-26.77, -49.83, -6.44) mm, rotated rx 180 ry 0 rz 90 deg; joints [71.941, -17.75, 85.25, 0, 22.5, 71.941]
  MoveL 4828 to (-25.92, -48.57, -6.84) mm, rotated rx -180 ry 0 rz 90 deg; joints [71.99, -17.721, 85.206, 0, 22.515, 71.99]
  MoveL 4829 to (-25.41, -47.14, -7.25) mm, rotated rx 180 ry 0 rz 90 deg; joints [72.042, -17.7, 85.189, 0, 22.511, 72.042]
  MoveL 4830 to (-19.66, -25.11, -7.25) mm, rotated rx 180 ry 0 rz 90 deg; joints [72.812, -17.721, 85.274, 0, 22.447, 72.812]
  MoveL 4831 to (-19.17, -23.22, -7.25) mm, rotated rx -180 ry 0 rz 90 deg; joints [72.878, -17.723, 85.281, 0, 22.442, 72.878]
  MoveL 4832 to (-19.06, -22.62, -7.25) mm, rotated rx 180 ry 0 rz 90 deg; joints [72.899, -17.724, 85.286, 0, 22.438, 72.899]
  MoveC 4833 to (-19.03, -21.94, -7.25) mm, rotated rx 180 ry 0 rz 90 deg; joints [72.921, -17.727, 85.298, 0, 22.429, 72.921] to (-19.19, -21.27, -7.25) mm, rotated rx -180 ry 0 rz 90 deg; joints [72.941, -17.734, 85.324, 0, 22.41, 72.941]
  MoveL 4834 to (-19.35, -20.88, -7.25) mm, rotated rx 180 ry 0 rz 90 deg; joints [72.952, -17.739, 85.344, 0, 22.395, 72.952]
  MoveC 4835 to (-20.69, -19.13, -7.25) mm, rotated rx -180 ry 0 rz 90 deg; joints [72.996, -17.772, 85.475, 0, 22.297, 72.996] to (-22.74, -18.33, -7.25) mm, rotated rx 180 ry 0 rz 90 deg; joints [73.001, -17.812, 85.635, 0, 22.178, 73.001]
  MoveL 4836 to (-23.22, -18.38, -7.25) mm, rotated rx -180 ry 0 rz 90 deg; joints [72.995, -17.82, 85.667, 0, 22.154, 72.995]
  MoveL 4837 to (-26.06, -18.97, -7.25) mm, rotated rx 180 ry 0 rz 90 deg; joints [72.947, -17.867, 85.852, 0, 22.015, 72.947]
  MoveL 4838 to (-71.94, -28.73, -7.25) mm, rotated rx 180 ry 0 rz 90 deg; joints [72.152, -18.568, 88.773, 0, 19.794, 72.152]
  MoveC 4839 to (-72.61, -28.92, -7.25) mm, rotated rx -180 ry 0 rz 90 deg; joints [72.139, -18.577, 88.814, 0, 19.763, 72.139] to (-73.24, -29.19, -7.25) mm, rotated rx 180 ry 0 rz 90 deg; joints [72.123, -18.585, 88.851, 0, 19.735, 72.123]
  MoveC 4840 to (-74.66, -30.5, -7.25) mm, rotated rx -180 ry 0 rz 90 deg; joints [72.064, -18.6, 88.917, 0, 19.683, 72.064] to (-75.18, -32.35, -7.25) mm, rotated rx 180 ry 0 rz 90 deg; joints [71.997, -18.599, 88.912, 0, 19.688, 71.997]
  MoveL 4841 to (-75.18, -70.81, -7.25) mm, rotated rx -180 ry 0 rz 90 deg; joints [70.728, -18.398, 88.043, 0, 20.355, 70.728]
  MoveC 4842 to (-74.95, -72.13, -7.25) mm, rotated rx -180 ry 0 rz 90 deg; joints [70.688, -18.387, 87.997, 0, 20.39, 70.688] to (-74.28, -73.29, -7.25) mm, rotated rx -180 ry 0 rz 90 deg; joints [70.657, -18.37, 87.925, 0, 20.445, 70.657]
  MoveC 4843 to (-73.04, -74.19, -7.25) mm, rotated rx 180 ry 0 rz 90 deg; joints [70.642, -18.346, 87.821, 0, 20.525, 70.642] to (-71.55, -74.53, -7.25) mm, rotated rx 180 ry 0 rz 90 deg; joints [70.648, -18.32, 87.712, 0, 20.608, 70.648]
  MoveL 4844 to (-70.6, -74.54, -7.25) mm, rotated rx -180 ry 0 rz 90 deg; joints [70.659, -18.305, 87.648, 0, 20.657, 70.659]
  MoveL 4845 to (-35.3, -74.26, -7.25) mm, rotated rx 180 ry 0 rz 90 deg; joints [71.064, -17.714, 85.247, 0, 22.467, 71.064]
  MoveC 4846 to (-33.13, -73.52, -7.25) mm, rotated rx -180 ry 0 rz 90 deg; joints [71.111, -17.681, 85.115, 0, 22.566, 71.111] to (-31.82, -71.64, -7.25) mm, rotated rx -180 ry 0 rz 90 deg; joints [71.186, -17.669, 85.068, 0, 22.601, 71.186]
  MoveL 4847 to (-31.51, -70.6, -7.25) mm, rotated rx 180 ry 0 rz 90 deg; joints [71.223, -17.67, 85.071, 0, 22.598, 71.223]
  MoveL 4848 to (-28.07, -57.33, -7.25) mm, rotated rx -180 ry 0 rz 90 deg; joints [71.686, -17.687, 85.141, 0, 22.546, 71.686]
  MoveL 4849 to (-25.41, -47.14, -7.25) mm, rotated rx 180 ry 0 rz 90 deg; joints [72.042, -17.7, 85.189, 0, 22.511, 72.042]
  MoveL 4850 to (-32.71, -45.23, -7.25) mm, rotated rx 180 ry 0 rz 90 deg; joints [72.027, -17.838, 85.739, 0, 22.1, 72.027]
  MoveL 4851 to (-32.71, -45.23, -4.25) mm, rotated rx 180 ry 0 rz 90 deg; joints [72.027, -17.993, 85.84, 0, 22.153, 72.027]
  Establecer velocidad (1000.0 mm/s)
  MoveL 4852 to (-32.71, -45.23, 10) mm, rotated rx 180 ry 0 rz 90 deg; joints [72.027, -18.725, 86.315, 0, 22.41, 72.027]
  Establecer velocidad (66.7 mm/s)
  MoveL 4853 to (-66.94, 36.36, 10) mm, rotated rx 180 ry 0 rz 90 deg; joints [74.388, -19.691, 90.328, 0, 19.363, 74.388]
  MoveL 4854 to (-66.94, 36.36, -4) mm, rotated rx -180 ry 0 rz 90 deg; joints [74.388, -18.958, 89.861, 0, 19.098, 74.388]
  MoveL 4855 to (-68.44, 36.55, -4.41) mm, rotated rx 180 ry 0 rz 90 deg; joints [74.38, -18.96, 89.952, 0, 19.009, 74.38]
  MoveL 4856 to (-69.95, 36.37, -4.81) mm, rotated rx -180 ry 0 rz 90 deg; joints [74.359, -18.961, 90.036, 0, 18.925, 74.359]
  MoveL 4857 to (-71.38, 35.85, -5.22) mm, rotated rx -180 ry 0 rz 90 deg; joints [74.328, -18.958, 90.108, 0, 18.85, 74.328]
  MoveL 4858 to (-72.66, 35.04, -5.63) mm, rotated rx 180 ry 0 rz 90 deg; joints [74.288, -18.953, 90.165, 0, 18.788, 74.288]
  MoveL 4859 to (-73.73, 33.96, -6.03) mm, rotated rx 180 ry 0 rz 90 deg; joints [74.241, -18.942, 90.202, 0, 18.74, 74.241]
  MoveL 4860 to (-74.54, 32.67, -6.44) mm, rotated rx -180 ry 0 rz 90 deg; joints [74.19, -18.928, 90.218, 0, 18.71, 74.19]
  MoveL 4861 to (-75.04, 31.23, -6.84) mm, rotated rx 180 ry 0 rz 90 deg; joints [74.136, -18.908, 90.21, 0, 18.697, 74.136]
  MoveL 4862 to (-75.18, 29.72, -7.25) mm, rotated rx 180 ry 0 rz 90 deg; joints [74.083, -18.882, 90.177, 0, 18.705, 74.083]
  MoveL 4863 to (-75.18, 1.42, -7.25) mm, rotated rx 180 ry 0 rz 90 deg; joints [73.126, -18.759, 89.621, 0, 19.138, 73.126]
  MoveL 4864 to (-75.16, 0.57, -7.25) mm, rotated rx -180 ry 0 rz 90 deg; joints [73.098, -18.755, 89.602, 0, 19.153, 73.098]
  MoveC 4865 to (-74.13, -1.88, -7.25) mm, rotated rx -180 ry 0 rz 90 deg; joints [73.026, -18.729, 89.484, 0, 19.245, 73.026] to (-71.72, -2.96, -7.25) mm, rotated rx 180 ry 0 rz 90 deg; joints [73.015, -18.687, 89.3, 0, 19.387, 73.015]
  MoveC 4866 to (-71.04, -2.95, -7.25) mm, rotated rx -180 ry 0 rz 90 deg; joints [73.022, -18.677, 89.255, 0, 19.422, 73.022] to (-70.37, -2.84, -7.25) mm, rotated rx -180 ry 0 rz 90 deg; joints [73.032, -18.668, 89.213, 0, 19.455, 73.032]
  MoveC 4867 to (-45.68, 2.82, -7.25) mm, rotated rx 180 ry 0 rz 90 deg; joints [73.469, -18.307, 87.656, 0, 20.65, 73.469] to (-20.99, 8.51, -7.25) mm, rotated rx 180 ry 0 rz 90 deg; joints [73.894, -17.921, 86.068, 0, 21.853, 73.894]
  MoveC 4868 to (-18.56, 10.33, -7.25) mm, rotated rx -180 ry 0 rz 90 deg; joints [73.977, -17.888, 85.936, 0, 21.952, 73.977] to (-18.29, 13.35, -7.25) mm, rotated rx 180 ry 0 rz 90 deg; joints [74.078, -17.898, 85.977, 0, 21.921, 74.078]
  MoveL 4869 to (-18.74, 14.69, -7.25) mm, rotated rx 180 ry 0 rz 90 deg; joints [74.118, -17.912, 86.035, 0, 21.877, 74.118]
  MoveL 4870 to (-24.52, 30.8, -7.25) mm, rotated rx -180 ry 0 rz 90 deg; joints [74.595, -18.089, 86.751, 0, 21.338, 74.595]
  MoveL 4871 to (-25.11, 32.4, -7.25) mm, rotated rx 180 ry 0 rz 90 deg; joints [74.643, -18.106, 86.823, 0, 21.284, 74.643]
  MoveL 4872 to (-25.17, 32.55, -7.25) mm, rotated rx -180 ry 0 rz 90 deg; joints [74.647, -18.108, 86.829, 0, 21.279, 74.647]
  MoveC 4873 to (-25.72, 33.5, -7.25) mm, rotated rx -180 ry 0 rz 90 deg; joints [74.674, -18.122, 86.886, 0, 21.236, 74.674] to (-26.54, 34.24, -7.25) mm, rotated rx 180 ry 0 rz 90 deg; joints [74.691, -18.139, 86.956, 0, 21.182, 74.691]
  MoveL 4874 to (-27.96, 35.18, -7.25) mm, rotated rx -180 ry 0 rz 90 deg; joints [74.709, -18.167, 87.072, 0, 21.095, 74.709]
  MoveL 4875 to (-64.01, 58.28, -7.25) mm, rotated rx 180 ry 0 rz 90 deg; joints [75.16, -18.833, 89.955, 0, 18.879, 75.16]
  MoveL 4876 to (-68.7, 61.3, -7.25) mm, rotated rx -180 ry 0 rz 90 deg; joints [75.221, -18.914, 90.324, 0, 18.59, 75.221]
  MoveC 4877 to (-69.62, 61.83, -7.25) mm, rotated rx -180 ry 0 rz 90 deg; joints [75.23, -18.929, 90.394, 0, 18.535, 75.23] to (-70.6, 62.22, -7.25) mm, rotated rx -180 ry 0 rz 90 deg; joints [75.235, -18.945, 90.467, 0, 18.478, 75.235]
  MoveC 4878 to (-73.29, 61.74, -7.25) mm, rotated rx 180 ry 0 rz 90 deg; joints [75.194, -18.982, 90.638, 0, 18.344, 75.194] to (-75.06, 59.66, -7.25) mm, rotated rx 180 ry 0 rz 90 deg; joints [75.107, -19, 90.72, 0, 18.28, 75.107]
  MoveC 4879 to (-75.14, 59.27, -7.25) mm, rotated rx -180 ry 0 rz 90 deg; joints [75.093, -18.999, 90.718, 0, 18.281, 75.093] to (-75.17, 58.88, -7.25) mm, rotated rx 180 ry 0 rz 90 deg; joints [75.079, -18.998, 90.713, 0, 18.286, 75.079]
  MoveL 4880 to (-75.18, 57.33, -7.25) mm, rotated rx 180 ry 0 rz 90 deg; joints [75.026, -18.992, 90.686, 0, 18.307, 75.026]
  MoveL 4881 to (-75.18, 29.72, -7.25) mm, rotated rx 180 ry 0 rz 90 deg; joints [74.083, -18.882, 90.177, 0, 18.705, 74.083]
  MoveL 4882 to (-67.63, 29.72, -7.25) mm, rotated rx 180 ry 0 rz 90 deg; joints [74.156, -18.771, 89.672, 0, 19.099, 74.156]
  MoveL 4883 to (-67.63, 29.72, -4.25) mm, rotated rx -180 ry 0 rz 90 deg; joints [74.156, -18.928, 89.773, 0, 19.154, 74.156]
  Establecer velocidad (1000.0 mm/s)
  MoveL 4884 to (-67.63, 29.72, 10) mm, rotated rx 180 ry 0 rz 90 deg; joints [74.156, -19.673, 90.249, 0, 19.424, 74.156]
  Establecer velocidad (66.7 mm/s)
  MoveL 4885 to (-66.76, 36.36, 10) mm, rotated rx -180 ry 0 rz 90 deg; joints [74.389, -19.688, 90.316, 0, 19.372, 74.389]
  MoveL 4886 to (-66.76, 36.36, -4.25) mm, rotated rx 180 ry 0 rz 90 deg; joints [74.389, -18.943, 89.841, 0, 19.102, 74.389]
  MoveL 4887 to (-68.27, 36.55, -4.66) mm, rotated rx 180 ry 0 rz 90 deg; joints [74.381, -18.945, 89.932, 0, 19.013, 74.381]
  MoveL 4888 to (-69.78, 36.37, -5.06) mm, rotated rx 180 ry 0 rz 90 deg; joints [74.361, -18.945, 90.016, 0, 18.929, 74.361]
  MoveL 4889 to (-71.21, 35.85, -5.47) mm, rotated rx -180 ry 0 rz 90 deg; joints [74.33, -18.943, 90.088, 0, 18.855, 74.33]
  MoveL 4890 to (-72.49, 35.04, -5.88) mm, rotated rx -180 ry 0 rz 90 deg; joints [74.29, -18.937, 90.145, 0, 18.792, 74.29]
  MoveL 4891 to (-73.56, 33.96, -6.28) mm, rotated rx 180 ry 0 rz 90 deg; joints [74.243, -18.927, 90.182, 0, 18.745, 74.243]
  MoveL 4892 to (-74.37, 32.67, -6.69) mm, rotated rx -180 ry 0 rz 90 deg; joints [74.191, -18.912, 90.198, 0, 18.714, 74.191]
  MoveL 4893 to (-74.87, 31.23, -7.09) mm, rotated rx 180 ry 0 rz 90 deg; joints [74.138, -18.892, 90.19, 0, 18.702, 74.138]
  MoveL 4894 to (-75, 29.72, -7.5) mm, rotated rx 180 ry 0 rz 90 deg; joints [74.085, -18.866, 90.157, 0, 18.71, 74.085]
  MoveL 4895 to (-75, 0.76, -7.5) mm, rotated rx 180 ry 0 rz 90 deg; joints [73.106, -18.741, 89.588, 0, 19.153, 73.106]
  MoveC 4896 to (-74.8, -0.4, -7.5) mm, rotated rx 180 ry 0 rz 90 deg; joints [73.069, -18.732, 89.55, 0, 19.182, 73.069] to (-74.22, -1.42, -7.5) mm, rotated rx -180 ry 0 rz 90 deg; joints [73.041, -18.719, 89.491, 0, 19.228, 73.041]
  MoveC 4897 to (-72.59, -2.57, -7.5) mm, rotated rx 180 ry 0 rz 90 deg; joints [73.019, -18.689, 89.358, 0, 19.331, 73.019] to (-70.6, -2.71, -7.5) mm, rotated rx -180 ry 0 rz 90 deg; joints [73.034, -18.659, 89.222, 0, 19.437, 73.034]
  MoveC 4898 to (-45.87, 2.96, -7.5) mm, rotated rx 180 ry 0 rz 90 deg; joints [73.472, -18.298, 87.664, 0, 20.634, 73.472] to (-21.14, 8.66, -7.5) mm, rotated rx 180 ry 0 rz 90 deg; joints [73.898, -17.911, 86.073, 0, 21.838, 73.898]
  MoveC 4899 to (-18.74, 10.47, -7.5) mm, rotated rx -180 ry 0 rz 90 deg; joints [73.98, -17.879, 85.943, 0, 21.936, 73.98] to (-18.51, 13.47, -7.5) mm, rotated rx 180 ry 0 rz 90 deg; joints [74.08, -17.889, 85.986, 0, 21.903, 74.08]
  MoveL 4900 to (-25.05, 31.75, -7.5) mm, rotated rx 180 ry 0 rz 90 deg; joints [74.622, -18.089, 86.797, 0, 21.292, 74.622]
  MoveL 4901 to (-25.36, 32.53, -7.5) mm, rotated rx 180 ry 0 rz 90 deg; joints [74.645, -18.098, 86.834, 0, 21.264, 74.645]
  MoveC 4902 to (-25.92, 33.46, -7.5) mm, rotated rx -180 ry 0 rz 90 deg; joints [74.671, -18.112, 86.89, 0, 21.222, 74.671] to (-26.72, 34.17, -7.5) mm, rotated rx 180 ry 0 rz 90 deg; joints [74.687, -18.129, 86.959, 0, 21.169, 74.687]
  MoveL 4903 to (-69.16, 61.37, -7.5) mm, rotated rx -180 ry 0 rz 90 deg; joints [75.219, -18.908, 90.347, 0, 18.561, 75.219]
  MoveC 4904 to (-69.85, 61.75, -7.5) mm, rotated rx -180 ry 0 rz 90 deg; joints [75.225, -18.919, 90.4, 0, 18.519, 75.225] to (-70.6, 62, -7.5) mm, rotated rx 180 ry 0 rz 90 deg; joints [75.227, -18.931, 90.454, 0, 18.477, 75.227]
  MoveC 4905 to (-73.28, 61.41, -7.5) mm, rotated rx 180 ry 0 rz 90 deg; joints [75.183, -18.968, 90.623, 0, 18.344, 75.183] to (-74.95, 59.23, -7.5) mm, rotated rx 180 ry 0 rz 90 deg; joints [75.093, -18.983, 90.696, 0, 18.287, 75.093]
  MoveL 4906 to (-75, 57.33, -7.5) mm, rotated rx 180 ry 0 rz 90 deg; joints [75.027, -18.977, 90.666, 0, 18.311, 75.027]
  MoveL 4907 to (-75, 29.72, -7.5) mm, rotated rx 180 ry 0 rz 90 deg; joints [74.085, -18.866, 90.157, 0, 18.71, 74.085]
  MoveL 4908 to (-67.45, 29.72, -7.5) mm, rotated rx 180 ry 0 rz 90 deg; joints [74.158, -18.755, 89.652, 0, 19.103, 74.158]
  MoveL 4909 to (-67.45, 29.72, -4.5) mm, rotated rx -180 ry 0 rz 90 deg; joints [74.158, -18.912, 89.753, 0, 19.159, 74.158]
  Establecer velocidad (1000.0 mm/s)
  MoveL 4910 to (-67.45, 29.72, 10) mm, rotated rx 180 ry 0 rz 90 deg; joints [74.158, -19.671, 90.237, 0, 19.433, 74.158]
  Establecer velocidad (66.7 mm/s)
  MoveL 4911 to (-39.86, -30.51, 10) mm, rotated rx 180 ry 0 rz 90 deg; joints [72.431, -18.931, 87.134, 0, 21.797, 72.431]
  MoveL 4912 to (-39.86, -30.51, -4.25) mm, rotated rx -180 ry 0 rz 90 deg; joints [72.431, -18.196, 86.659, 0, 21.538, 72.431]
  MoveL 4913 to (-39.99, -29, -4.66) mm, rotated rx 180 ry 0 rz 90 deg; joints [72.479, -18.186, 86.687, 0, 21.499, 72.479]
  MoveL 4914 to (-40.49, -27.56, -5.06) mm, rotated rx 180 ry 0 rz 90 deg; joints [72.521, -18.181, 86.738, 0, 21.443, 72.521]
  MoveL 4915 to (-41.29, -26.27, -5.47) mm, rotated rx 180 ry 0 rz 90 deg; joints [72.555, -18.18, 86.807, 0, 21.373, 72.555]
  MoveL 4916 to (-42.35, -25.18, -5.88) mm, rotated rx -180 ry 0 rz 90 deg; joints [72.579, -18.182, 86.89, 0, 21.293, 72.579]
  MoveL 4917 to (-43.63, -24.36, -6.28) mm, rotated rx 180 ry 0 rz 90 deg; joints [72.593, -18.187, 86.981, 0, 21.206, 72.593]
  MoveL 4918 to (-45.05, -23.85, -6.69) mm, rotated rx -180 ry 0 rz 90 deg; joints [72.595, -18.192, 87.076, 0, 21.116, 72.595]
  MoveL 4919 to (-46.56, -23.66, -7.09) mm, rotated rx 180 ry 0 rz 90 deg; joints [72.586, -18.197, 87.17, 0, 21.027, 72.586]
  MoveL 4920 to (-48.07, -23.83, -7.5) mm, rotated rx 180 ry 0 rz 90 deg; joints [72.565, -18.2, 87.255, 0, 20.945, 72.565]
  MoveC 4921 to (-60.03, -26.38, -7.5) mm, rotated rx -180 ry 0 rz 90 deg; joints [72.356, -18.38, 88.013, 0, 20.367, 72.356] to (-71.99, -28.94, -7.5) mm, rotated rx 180 ry 0 rz 90 deg; joints [72.145, -18.554, 88.764, 0, 19.791, 72.145]
  MoveC 4922 to (-72.39, -29.04, -7.5) mm, rotated rx -180 ry 0 rz 90 deg; joints [72.137, -18.56, 88.788, 0, 19.772, 72.137] to (-72.77, -29.17, -7.5) mm, rotated rx -180 ry 0 rz 90 deg; joints [72.129, -18.565, 88.811, 0, 19.754, 72.129]
  MoveC 4923 to (-74.39, -30.45, -7.5) mm, rotated rx 180 ry 0 rz 90 deg; joints [72.068, -18.584, 88.892, 0, 19.692, 72.068] to (-75, -32.43, -7.5) mm, rotated rx -180 ry 0 rz 90 deg; joints [71.996, -18.583, 88.89, 0, 19.693, 71.996]
  MoveL 4924 to (-75, -70.8, -7.5) mm, rotated rx 180 ry 0 rz 90 deg; joints [70.731, -18.382, 88.023, 0, 20.359, 70.731]
  MoveC 4925 to (-73.99, -73.28, -7.5) mm, rotated rx 180 ry 0 rz 90 deg; joints [70.661, -18.353, 87.897, 0, 20.455, 70.661] to (-71.53, -74.34, -7.5) mm, rotated rx 180 ry 0 rz 90 deg; joints [70.655, -18.308, 87.707, 0, 20.601, 70.655]
  MoveL 4926 to (-70.6, -74.36, -7.5) mm, rotated rx 180 ry 0 rz 90 deg; joints [70.665, -18.293, 87.644, 0, 20.649, 70.665]
  MoveL 4927 to (-64.91, -74.32, -7.5) mm, rotated rx 180 ry 0 rz 90 deg; joints [70.731, -18.202, 87.262, 0, 20.94, 70.731]
  MoveL 4928 to (-35.38, -74.09, -7.5) mm, rotated rx -180 ry 0 rz 90 deg; joints [71.069, -17.704, 85.248, 0, 22.456, 71.069]
  MoveC 4929 to (-33.22, -73.35, -7.5) mm, rotated rx 180 ry 0 rz 90 deg; joints [71.116, -17.67, 85.117, 0, 22.554, 71.116] to (-31.95, -71.46, -7.5) mm, rotated rx -180 ry 0 rz 90 deg; joints [71.19, -17.659, 85.073, 0, 22.586, 71.19]
  MoveL 4930 to (-31.71, -70.6, -7.5) mm, rotated rx -180 ry 0 rz 90 deg; joints [71.221, -17.66, 85.077, 0, 22.584, 71.221]
  MoveL 4931 to (-21.17, -30.18, -7.5) mm, rotated rx -180 ry 0 rz 90 deg; joints [72.633, -17.707, 85.261, 0, 22.446, 72.633]
  MoveC 4932 to (-20.25, -26.63, -7.5) mm, rotated rx 180 ry 0 rz 90 deg; joints [72.757, -17.71, 85.274, 0, 22.436, 72.757] to (-19.33, -23.07, -7.5) mm, rotated rx 180 ry 0 rz 90 deg; joints [72.881, -17.714, 85.287, 0, 22.427, 72.881]
  MoveC 4933 to (-19.24, -22.23, -7.5) mm, rotated rx 180 ry 0 rz 90 deg; joints [72.91, -17.717, 85.299, 0, 22.418, 72.91] to (-19.41, -21.4, -7.5) mm, rotated rx 180 ry 0 rz 90 deg; joints [72.935, -17.724, 85.328, 0, 22.396, 72.935]
  MoveC 4934 to (-20.52, -19.69, -7.5) mm, rotated rx 180 ry 0 rz 90 deg; joints [72.979, -17.753, 85.442, 0, 22.311, 72.979] to (-22.27, -18.65, -7.5) mm, rotated rx -180 ry 0 rz 90 deg; joints [72.996, -17.789, 85.587, 0, 22.203, 72.996]
  MoveC 4935 to (-22.8, -18.55, -7.5) mm, rotated rx -180 ry 0 rz 90 deg; joints [72.993, -17.799, 85.626, 0, 22.174, 72.993] to (-23.34, -18.6, -7.5) mm, rotated rx 180 ry 0 rz 90 deg; joints [72.987, -17.808, 85.662, 0, 22.146, 72.987]
  MoveC 4936 to (-35.71, -21.21, -7.5) mm, rotated rx 180 ry 0 rz 90 deg; joints [72.777, -18.007, 86.463, 0, 21.544, 72.777] to (-48.07, -23.83, -7.5) mm, rotated rx -180 ry 0 rz 90 deg; joints [72.565, -18.2, 87.255, 0, 20.945, 72.565]
  MoveL 4937 to (-46.5, -31.22, -7.5) mm, rotated rx -180 ry 0 rz 90 deg; joints [72.339, -18.136, 86.988, 0, 21.147, 72.339]
  MoveL 4938 to (-46.5, -31.22, -4.5) mm, rotated rx -180 ry 0 rz 90 deg; joints [72.339, -18.291, 87.09, 0, 21.201, 72.339]
  Establecer velocidad (1000.0 mm/s)
  MoveL 4939 to (-46.5, -31.22, 10) mm, rotated rx 180 ry 0 rz 90 deg; joints [72.339, -19.04, 87.574, 0, 21.466, 72.339]
  Establecer velocidad (66.7 mm/s)
  MoveL 4940 to (15.55, -65.72, 10) mm, rotated rx 180 ry 0 rz 90 deg; joints [71.875, -17.69, 82.436, 0, 25.254, 71.875]
  MoveL 4941 to (15.55, -65.72, -4.25) mm, rotated rx 180 ry 0 rz 90 deg; joints [71.875, -16.969, 81.959, 0, 25.01, 71.875]
  MoveL 4942 to (15.4, -67.23, -4.66) mm, rotated rx -180 ry 0 rz 90 deg; joints [71.826, -16.942, 81.92, 0, 25.021, 71.826]
  MoveL 4943 to (15.61, -68.73, -5.06) mm, rotated rx -180 ry 0 rz 90 deg; joints [71.781, -16.907, 81.856, 0, 25.051, 71.781]
  MoveL 4944 to (16.14, -70.16, -5.47) mm, rotated rx 180 ry 0 rz 90 deg; joints [71.742, -16.866, 81.769, 0, 25.097, 71.742]
  MoveL 4945 to (16.98, -71.42, -5.88) mm, rotated rx 180 ry 0 rz 90 deg; joints [71.711, -16.821, 81.665, 0, 25.156, 71.711]
  MoveL 4946 to (18.08, -72.48, -6.28) mm, rotated rx -180 ry 0 rz 90 deg; joints [71.69, -16.771, 81.547, 0, 25.225, 71.69]
  MoveL 4947 to (19.38, -73.26, -6.69) mm, rotated rx 180 ry 0 rz 90 deg; joints [71.679, -16.719, 81.42, 0, 25.3, 71.679]
  MoveL 4948 to (20.83, -73.73, -7.09) mm, rotated rx -180 ry 0 rz 90 deg; joints [71.679, -16.666, 81.29, 0, 25.377, 71.679]
  MoveL 4949 to (22.34, -73.84, -7.5) mm, rotated rx 180 ry 0 rz 90 deg; joints [71.691, -16.615, 81.163, 0, 25.451, 71.691]
  MoveC 4950 to (35.06, -73.59, -7.5) mm, rotated rx 180 ry 0 rz 90 deg; joints [71.829, -16.355, 80.24, 0, 26.115, 71.829] to (47.79, -73.3, -7.5) mm, rotated rx -180 ry 0 rz 90 deg; joints [71.966, -16.087, 79.307, 0, 26.78, 71.966]
  MoveC 4951 to (50.4, -70.25, -7.5) mm, rotated rx 180 ry 0 rz 90 deg; joints [72.086, -16.052, 79.186, 0, 26.866, 72.086] to (50.54, -66.24, -7.5) mm, rotated rx 180 ry 0 rz 90 deg; joints [72.211, -16.077, 79.272, 0, 26.805, 72.211]
  MoveL 4952 to (48.63, -63.97, -7.5) mm, rotated rx 180 ry 0 rz 90 deg; joints [72.263, -16.134, 79.468, 0, 26.666, 72.263]
  MoveL 4953 to (30.09, -42.17, -7.5) mm, rotated rx -180 ry 0 rz 90 deg; joints [72.759, -16.663, 81.338, 0, 25.325, 72.759]
  MoveL 4954 to (27.01, -38.59, -7.5) mm, rotated rx 180 ry 0 rz 90 deg; joints [72.842, -16.748, 81.644, 0, 25.104, 72.842]
  MoveL 4955 to (25.17, -36.48, -7.5) mm, rotated rx -180 ry 0 rz 90 deg; joints [72.891, -16.798, 81.824, 0, 24.974, 72.891]
  MoveL 4956 to (25.11, -36.43, -7.5) mm, rotated rx -180 ry 0 rz 90 deg; joints [72.892, -16.799, 81.83, 0, 24.97, 72.892]
  MoveL 4957 to (24.02, -35.54, -7.5) mm, rotated rx 180 ry 0 rz 90 deg; joints [72.909, -16.826, 81.929, 0, 24.897, 72.909]
  MoveL 4958 to (12.1, -25.97, -7.5) mm, rotated rx -180 ry 0 rz 90 deg; joints [73.097, -17.117, 82.999, 0, 24.117, 73.097]
  MoveC 4959 to (9.27, -25.59, -7.5) mm, rotated rx -180 ry 0 rz 90 deg; joints [73.082, -17.173, 83.21, 0, 23.963, 73.082] to (6.8, -27.01, -7.5) mm, rotated rx 180 ry 0 rz 90 deg; joints [73.013, -17.212, 83.356, 0, 23.856, 73.013]
  MoveC 4960 to (6.49, -27.48, -7.5) mm, rotated rx -180 ry 0 rz 90 deg; joints [72.995, -17.215, 83.368, 0, 23.847, 72.995] to (6.29, -28, -7.5) mm, rotated rx -180 ry 0 rz 90 deg; joints [72.976, -17.216, 83.371, 0, 23.845, 72.976]
  MoveL 4961 to (-4.59, -68.7, -7.5) mm, rotated rx 180 ry 0 rz 90 deg; joints [71.572, -17.175, 83.219, 0, 23.957, 71.572]
  MoveL 4962 to (-4.77, -69.43, -7.5) mm, rotated rx 180 ry 0 rz 90 deg; joints [71.547, -17.174, 83.215, 0, 23.96, 71.547]
  MoveC 4963 to (-4.59, -71.83, -7.5) mm, rotated rx -180 ry 0 rz 90 deg; joints [71.473, -17.156, 83.145, 0, 24.011, 71.473] to (-2.99, -73.61, -7.5) mm, rotated rx 180 ry 0 rz 90 deg; joints [71.433, -17.114, 82.989, 0, 24.125, 71.433]
  MoveL 4964 to (-2.37, -73.96, -7.5) mm, rotated rx 180 ry 0 rz 90 deg; joints [71.429, -17.1, 82.936, 0, 24.164, 71.429]
  MoveL 4965 to (-1.42, -74.19, -7.5) mm, rotated rx -180 ry 0 rz 90 deg; joints [71.432, -17.08, 82.864, 0, 24.217, 71.432]
  MoveC 4966 to (10.46, -74.03, -7.5) mm, rotated rx 180 ry 0 rz 90 deg; joints [71.562, -16.851, 82.017, 0, 24.833, 71.562] to (22.34, -73.84, -7.5) mm, rotated rx 180 ry 0 rz 90 deg; joints [71.691, -16.615, 81.163, 0, 25.451, 71.691]
  MoveL 4967 to (22.21, -66.29, -7.5) mm, rotated rx 180 ry 0 rz 90 deg; joints [71.925, -16.667, 81.353, 0, 25.314, 71.925]
  MoveL 4968 to (22.21, -66.29, -4.5) mm, rotated rx 180 ry 0 rz 90 deg; joints [71.925, -16.819, 81.455, 0, 25.364, 71.925]
  Establecer velocidad (1000.0 mm/s)
  MoveL 4969 to (22.21, -66.29, 10) mm, rotated rx -180 ry 0 rz 90 deg; joints [71.925, -17.552, 81.941, 0, 25.61, 71.925]
  Establecer velocidad (66.7 mm/s)
  MoveL 4970 to (63.69, -31.17, 10) mm, rotated rx -180 ry 0 rz 90 deg; joints [73.421, -16.905, 79.691, 0, 27.214, 73.421]
  MoveL 4971 to (63.69, -31.17, -4.25) mm, rotated rx 180 ry 0 rz 90 deg; joints [73.421, -16.191, 79.211, 0, 26.98, 73.421]
  MoveL 4972 to (65.19, -31.35, -4.66) mm, rotated rx 180 ry 0 rz 90 deg; joints [73.429, -16.136, 79.08, 0, 27.056, 73.429]
  MoveL 4973 to (66.7, -31.17, -5.06) mm, rotated rx -180 ry 0 rz 90 deg; joints [73.449, -16.084, 78.957, 0, 27.127, 73.449]
  MoveL 4974 to (68.13, -30.66, -5.47) mm, rotated rx 180 ry 0 rz 90 deg; joints [73.478, -16.035, 78.846, 0, 27.189, 73.478]
  MoveL 4975 to (69.41, -29.84, -5.88) mm, rotated rx 180 ry 0 rz 90 deg; joints [73.515, -15.992, 78.754, 0, 27.238, 73.515]
  MoveL 4976 to (70.48, -28.76, -6.28) mm, rotated rx 180 ry 0 rz 90 deg; joints [73.558, -15.955, 78.683, 0, 27.271, 73.558]
  MoveL 4977 to (71.29, -27.47, -6.69) mm, rotated rx 180 ry 0 rz 90 deg; joints [73.605, -15.925, 78.638, 0, 27.288, 73.605]
  MoveL 4978 to (71.79, -26.03, -7.09) mm, rotated rx 180 ry 0 rz 90 deg; joints [73.654, -15.903, 78.618, 0, 27.285, 73.654]
  MoveL 4979 to (71.93, -24.53, -7.5) mm, rotated rx 180 ry 0 rz 90 deg; joints [73.702, -15.889, 78.627, 0, 27.263, 73.702]
  MoveL 4980 to (71.93, -14.58, -7.5) mm, rotated rx -180 ry 0 rz 90 deg; joints [74.01, -15.953, 78.844, 0, 27.109, 74.01]
  MoveC 4981 to (69.53, -11.46, -7.5) mm, rotated rx 180 ry 0 rz 90 deg; joints [74.086, -16.025, 79.092, 0, 26.933, 74.086] to (65.81, -10.17, -7.5) mm, rotated rx -180 ry 0 rz 90 deg; joints [74.093, -16.114, 79.4, 0, 26.714, 74.093]
  MoveC 4982 to (65.16, -10.3, -7.5) mm, rotated rx 180 ry 0 rz 90 deg; joints [74.083, -16.127, 79.446, 0, 26.681, 74.083] to (64.64, -10.73, -7.5) mm, rotated rx 180 ry 0 rz 90 deg; joints [74.065, -16.136, 79.476, 0, 26.66, 74.065]
  MoveL 4983 to (55.46, -23.22, -7.5) mm, rotated rx 180 ry 0 rz 90 deg; joints [73.593, -16.255, 79.891, 0, 26.364, 73.593]
  MoveL 4984 to (54.99, -23.91, -7.5) mm, rotated rx -180 ry 0 rz 90 deg; joints [73.567, -16.261, 79.911, 0, 26.35, 73.567]
  MoveC 4985 to (54.38, -26.13, -7.5) mm, rotated rx 180 ry 0 rz 90 deg; joints [73.492, -16.26, 79.907, 0, 26.353, 73.492] to (55.27, -28.26, -7.5) mm, rotated rx -180 ry 0 rz 90 deg; joints [73.434, -16.227, 79.794, 0, 26.434, 73.434]
  MoveL 4986 to (65.34, -39.54, -7.5) mm, rotated rx -180 ry 0 rz 90 deg; joints [73.178, -15.936, 78.787, 0, 27.149, 73.178]
  MoveC 4987 to (68.24, -39.26, -7.5) mm, rotated rx -180 ry 0 rz 90 deg; joints [73.213, -15.874, 78.574, 0, 27.3, 73.213] to (70.6, -37.55, -7.5) mm, rotated rx 180 ry 0 rz 90 deg; joints [73.288, -15.833, 78.435, 0, 27.398, 73.288]
  MoveC 4988 to (71.58, -36.14, -7.5) mm, rotated rx 180 ry 0 rz 90 deg; joints [73.34, -15.821, 78.393, 0, 27.428, 73.34] to (71.93, -34.47, -7.5) mm, rotated rx 180 ry 0 rz 90 deg; joints [73.395, -15.824, 78.405, 0, 27.42, 73.395]
  MoveL 4989 to (71.93, -24.53, -7.5) mm, rotated rx 180 ry 0 rz 90 deg; joints [73.702, -15.889, 78.627, 0, 27.263, 73.702]
  MoveL 4990 to (64.38, -24.53, -7.5) mm, rotated rx -180 ry 0 rz 90 deg; joints [73.634, -16.055, 79.195, 0, 26.86, 73.634]
  MoveL 4991 to (64.38, -24.53, -4.5) mm, rotated rx 180 ry 0 rz 90 deg; joints [73.634, -16.206, 79.298, 0, 26.908, 73.634]
  Establecer velocidad (1000.0 mm/s)
  MoveL 4992 to (64.38, -24.53, 10) mm, rotated rx 180 ry 0 rz 90 deg; joints [73.634, -16.933, 79.786, 0, 27.147, 73.634]
  Establecer velocidad (66.7 mm/s)
  MoveL 4993 to (32.54, 9.45, 10) mm, rotated rx -180 ry 0 rz 90 deg; joints [74.416, -17.806, 82.855, 0, 24.951, 74.416]
  MoveL 4994 to (32.54, 9.45, -4.25) mm, rotated rx 180 ry 0 rz 90 deg; joints [74.416, -17.084, 82.378, 0, 24.706, 74.416]
  MoveL 4995 to (33.66, 8.43, -4.66) mm, rotated rx 180 ry 0 rz 90 deg; joints [74.393, -17.036, 82.262, 0, 24.773, 74.393]
  MoveL 4996 to (35, 7.7, -5.06) mm, rotated rx -180 ry 0 rz 90 deg; joints [74.382, -16.984, 82.136, 0, 24.848, 74.382]
  MoveL 4997 to (36.46, 7.29, -5.47) mm, rotated rx -180 ry 0 rz 90 deg; joints [74.382, -16.932, 82.007, 0, 24.925, 74.382]
  MoveL 4998 to (37.98, 7.22, -5.88) mm, rotated rx 180 ry 0 rz 90 deg; joints [74.393, -16.88, 81.881, 0, 24.999, 74.393]
  MoveL 4999 to (39.47, 7.48, -6.28) mm, rotated rx -180 ry 0 rz 90 deg; joints [74.415, -16.831, 81.763, 0, 25.068, 74.415]
  MoveL 5000 to (40.88, 8.07, -6.69) mm, rotated rx -180 ry 0 rz 90 deg; joints [74.446, -16.785, 81.658, 0, 25.127, 74.446]
  MoveL 5001 to (42.11, 8.95, -7.09) mm, rotated rx -180 ry 0 rz 90 deg; joints [74.485, -16.745, 81.572, 0, 25.173, 74.485]
  MoveL 5002 to (43.1, 10.11, -7.5) mm, rotated rx -180 ry 0 rz 90 deg; joints [74.53, -16.711, 81.509, 0, 25.202, 74.53]
  MoveL 5003 to (52.04, 22.74, -7.5) mm, rotated rx 180 ry 0 rz 90 deg; joints [75.008, -16.598, 81.103, 0, 25.494, 75.008]
  MoveL 5004 to (52.12, 22.89, -7.5) mm, rotated rx -180 ry 0 rz 90 deg; joints [75.013, -16.597, 81.1, 0, 25.497, 75.013]
  MoveC 5005 to (51.88, 26.42, -7.5) mm, rotated rx -180 ry 0 rz 90 deg; joints [75.123, -16.621, 81.188, 0, 25.433, 75.123] to (49.73, 29.24, -7.5) mm, rotated rx -180 ry 0 rz 90 deg; joints [75.195, -16.681, 81.402, 0, 25.279, 75.195]
  MoveC 5006 to (49.2, 29.5, -7.5) mm, rotated rx -180 ry 0 rz 90 deg; joints [75.199, -16.693, 81.446, 0, 25.247, 75.199] to (48.62, 29.59, -7.5) mm, rotated rx 180 ry 0 rz 90 deg; joints [75.197, -16.706, 81.49, 0, 25.215, 75.197]
  MoveC 5007 to (29.29, 29.28, -7.5) mm, rotated rx 180 ry 0 rz 90 deg; joints [75.022, -17.09, 82.898, 0, 24.192, 75.022] to (9.95, 28.88, -7.5) mm, rotated rx 180 ry 0 rz 90 deg; joints [74.841, -17.455, 84.281, 0, 23.175, 74.841]
  MoveC 5008 to (7.26, 27.24, -7.5) mm, rotated rx -180 ry 0 rz 90 deg; joints [74.764, -17.497, 84.44, 0, 23.056, 74.764] to (6.55, 24.17, -7.5) mm, rotated rx 180 ry 0 rz 90 deg; joints [74.658, -17.494, 84.431, 0, 23.063, 74.658]
  MoveL 5009 to (6.72, 23.67, -7.5) mm, rotated rx 180 ry 0 rz 90 deg; joints [74.643, -17.489, 84.409, 0, 23.079, 74.643]
  MoveL 5010 to (11.72, 9.95, -7.5) mm, rotated rx 180 ry 0 rz 90 deg; joints [74.245, -17.324, 83.78, 0, 23.544, 74.245]
  MoveL 5011 to (11.93, 9.43, -7.5) mm, rotated rx 180 ry 0 rz 90 deg; joints [74.23, -17.318, 83.755, 0, 23.563, 74.23]
  MoveC 5012 to (12.38, 8.62, -7.5) mm, rotated rx 180 ry 0 rz 90 deg; joints [74.208, -17.305, 83.706, 0, 23.599, 74.208] to (13.03, 7.97, -7.5) mm, rotated rx -180 ry 0 rz 90 deg; joints [74.193, -17.289, 83.646, 0, 23.643, 74.193]
  MoveL 5013 to (27.96, -3.49, -7.5) mm, rotated rx 180 ry 0 rz 90 deg; joints [73.962, -16.937, 82.335, 0, 24.603, 73.962]
  MoveL 5014 to (28.9, -4.16, -7.5) mm, rotated rx -180 ry 0 rz 90 deg; joints [73.95, -16.915, 82.252, 0, 24.663, 73.95]
  MoveC 5015 to (31.74, -4.31, -7.5) mm, rotated rx -180 ry 0 rz 90 deg; joints [73.971, -16.857, 82.042, 0, 24.815, 73.971] to (34.06, -2.66, -7.5) mm, rotated rx 180 ry 0 rz 90 deg; joints [74.044, -16.821, 81.908, 0, 24.913, 74.044]
  MoveL 5016 to (43.1, 10.11, -7.5) mm, rotated rx -180 ry 0 rz 90 deg; joints [74.53, -16.711, 81.509, 0, 25.202, 74.53]
  MoveL 5017 to (36.93, 14.47, -7.5) mm, rotated rx 180 ry 0 rz 90 deg; joints [74.615, -16.859, 82.049, 0, 24.81, 74.615]
  MoveL 5018 to (36.93, 14.47, -4.5) mm, rotated rx -180 ry 0 rz 90 deg; joints [74.615, -17.011, 82.151, 0, 24.861, 74.615]
  Establecer velocidad (1000.0 mm/s)
  MoveL 5019 to (36.93, 14.47, 10) mm, rotated rx 180 ry 0 rz 90 deg; joints [74.615, -17.746, 82.636, 0, 25.11, 74.615]
  Establecer velocidad (66.7 mm/s)
  MoveL 5020 to (27.75, 65.28, 10) mm, rotated rx 180 ry 0 rz 90 deg; joints [76.173, -18.189, 84.264, 0, 23.925, 76.173]
  MoveL 5021 to (27.75, 65.28, -4.25) mm, rotated rx 180 ry 0 rz 90 deg; joints [76.173, -17.463, 83.788, 0, 23.675, 76.173]
  MoveL 5022 to (27.96, 66.78, -4.66) mm, rotated rx 180 ry 0 rz 90 deg; joints [76.223, -17.446, 83.786, 0, 23.66, 76.223]
  MoveL 5023 to (27.81, 68.29, -5.06) mm, rotated rx -180 ry 0 rz 90 deg; joints [76.271, -17.435, 83.81, 0, 23.625, 76.271]
  MoveL 5024 to (27.32, 69.73, -5.47) mm, rotated rx -180 ry 0 rz 90 deg; joints [76.314, -17.43, 83.857, 0, 23.573, 76.314]
  MoveL 5025 to (26.53, 71.03, -5.88) mm, rotated rx -180 ry 0 rz 90 deg; joints [76.35, -17.43, 83.923, 0, 23.507, 76.35]
  MoveL 5026 to (25.47, 72.12, -6.28) mm, rotated rx 180 ry 0 rz 90 deg; joints [76.377, -17.435, 84.004, 0, 23.43, 76.377]
  MoveL 5027 to (24.2, 72.95, -6.69) mm, rotated rx 180 ry 0 rz 90 deg; joints [76.394, -17.442, 84.097, 0, 23.345, 76.394]
  MoveL 5028 to (22.77, 73.47, -7.09) mm, rotated rx -180 ry 0 rz 90 deg; joints [76.4, -17.45, 84.195, 0, 23.255, 76.4]
  MoveL 5029 to (21.26, 73.64, -7.5) mm, rotated rx -180 ry 0 rz 90 deg; joints [76.394, -17.458, 84.292, 0, 23.166, 76.394]
  MoveL 5030 to (12.79, 73.8, -7.5) mm, rotated rx 180 ry 0 rz 90 deg; joints [76.332, -17.615, 84.901, 0, 22.714, 76.332]
  MoveL 5031 to (-24.17, 74.33, -7.5) mm, rotated rx 180 ry 0 rz 90 deg; joints [76.048, -18.261, 87.508, 0, 20.752, 76.048]
  MoveL 5032 to (-25.91, 74.35, -7.5) mm, rotated rx -180 ry 0 rz 90 deg; joints [76.034, -18.289, 87.629, 0, 20.66, 76.034]
  MoveC 5033 to (-28.46, 71.14, -7.5) mm, rotated rx 180 ry 0 rz 90 deg; joints [75.905, -18.318, 87.75, 0, 20.568, 75.905] to (-28.05, 67.07, -7.5) mm, rotated rx -180 ry 0 rz 90 deg; joints [75.772, -18.294, 87.651, 0, 20.644, 75.772]
  MoveL 5034 to (-9.8, 55.44, -7.5) mm, rotated rx -180 ry 0 rz 90 deg; joints [75.54, -17.936, 86.174, 0, 21.762, 75.54]
  MoveC 5035 to (-8.51, 54.86, -7.5) mm, rotated rx 180 ry 0 rz 90 deg; joints [75.532, -17.911, 86.073, 0, 21.838, 75.532] to (-7.11, 54.75, -7.5) mm, rotated rx -180 ry 0 rz 90 deg; joints [75.541, -17.886, 85.973, 0, 21.914, 75.541]
  MoveL 5036 to (-3.32, 55.05, -7.5) mm, rotated rx 180 ry 0 rz 90 deg; joints [75.582, -17.821, 85.711, 0, 22.11, 75.582]
  MoveL 5037 to (21.32, 56.87, -7.5) mm, rotated rx 180 ry 0 rz 90 deg; joints [75.847, -17.379, 83.99, 0, 23.389, 75.847]
  MoveL 5038 to (26.06, 57.25, -7.5) mm, rotated rx -180 ry 0 rz 90 deg; joints [75.898, -17.291, 83.656, 0, 23.636, 75.898]
  MoveL 5039 to (28.9, 57.49, -7.5) mm, rotated rx 180 ry 0 rz 90 deg; joints [75.929, -17.238, 83.455, 0, 23.783, 75.929]
  MoveC 5040 to (45.51, 59.03, -7.5) mm, rotated rx -180 ry 0 rz 90 deg; joints [76.113, -16.921, 82.273, 0, 24.647, 76.113] to (62.07, 61, -7.5) mm, rotated rx 180 ry 0 rz 90 deg; joints [76.306, -16.593, 81.085, 0, 25.508, 76.306]
  MoveL 5041 to (62.94, 61.12, -7.5) mm, rotated rx -180 ry 0 rz 90 deg; joints [76.316, -16.575, 81.023, 0, 25.552, 76.316]
  MoveL 5042 to (68.52, 61.97, -7.5) mm, rotated rx -180 ry 0 rz 90 deg; joints [76.386, -16.463, 80.622, 0, 25.841, 76.386]
  MoveC 5043 to (70.09, 62.78, -7.5) mm, rotated rx -180 ry 0 rz 90 deg; joints [76.424, -16.434, 80.519, 0, 25.915, 76.424] to (70.82, 64.39, -7.5) mm, rotated rx -180 ry 0 rz 90 deg; joints [76.481, -16.426, 80.493, 0, 25.933, 76.481]
  MoveC 5044 to (70.94, 66.84, -7.5) mm, rotated rx 180 ry 0 rz 90 deg; joints [76.56, -16.436, 80.528, 0, 25.908, 76.56] to (70.82, 69.28, -7.5) mm, rotated rx -180 ry 0 rz 90 deg; joints [76.636, -16.451, 80.581, 0, 25.87, 76.636]
  MoveC 5045 to (70.04, 70.9, -7.5) mm, rotated rx -180 ry 0 rz 90 deg; joints [76.682, -16.476, 80.668, 0, 25.808, 76.682] to (68.4, 71.62, -7.5) mm, rotated rx 180 ry 0 rz 90 deg; joints [76.693, -16.514, 80.804, 0, 25.71, 76.693]
  MoveC 5046 to (44.84, 72.94, -7.5) mm, rotated rx 180 ry 0 rz 90 deg; joints [76.555, -17.001, 82.57, 0, 24.431, 76.555] to (21.26, 73.64, -7.5) mm, rotated rx -180 ry 0 rz 90 deg; joints [76.394, -17.458, 84.292, 0, 23.166, 76.394]
  MoveL 5047 to (21.12, 66.09, -7.5) mm, rotated rx 180 ry 0 rz 90 deg; joints [76.146, -17.426, 84.17, 0, 23.256, 76.146]
  MoveL 5048 to (21.12, 66.09, -4.5) mm, rotated rx 180 ry 0 rz 90 deg; joints [76.146, -17.58, 84.272, 0, 23.308, 76.146]
  Establecer velocidad (1000.0 mm/s)
  MoveL 5049 to (21.12, 66.09, 10) mm, rotated rx 180 ry 0 rz 90 deg; joints [76.146, -18.32, 84.756, 0, 23.564, 76.146]
  Establecer velocidad (66.7 mm/s)
  MoveL 5050 to (27.73, 65.03, 10) mm, rotated rx 180 ry 0 rz 90 deg; joints [76.165, -18.188, 84.261, 0, 23.927, 76.165]
  MoveL 5051 to (27.73, 65.03, -4.5) mm, rotated rx 180 ry 0 rz 90 deg; joints [76.165, -17.45, 83.777, 0, 23.673, 76.165]
  MoveL 5052 to (27.95, 66.53, -4.91) mm, rotated rx -180 ry 0 rz 90 deg; joints [76.215, -17.432, 83.774, 0, 23.658, 76.215]
  MoveL 5053 to (27.8, 68.04, -5.31) mm, rotated rx 180 ry 0 rz 90 deg; joints [76.263, -17.421, 83.798, 0, 23.623, 76.263]
  MoveL 5054 to (27.31, 69.48, -5.72) mm, rotated rx 180 ry 0 rz 90 deg; joints [76.306, -17.416, 83.845, 0, 23.572, 76.306]
  MoveL 5055 to (26.52, 70.78, -6.12) mm, rotated rx -180 ry 0 rz 90 deg; joints [76.342, -17.417, 83.911, 0, 23.506, 76.342]
  MoveL 5056 to (25.47, 71.87, -6.53) mm, rotated rx 180 ry 0 rz 90 deg; joints [76.369, -17.421, 83.992, 0, 23.429, 76.369]
  MoveL 5057 to (24.19, 72.7, -6.94) mm, rotated rx 180 ry 0 rz 90 deg; joints [76.386, -17.428, 84.085, 0, 23.343, 76.386]
  MoveL 5058 to (22.77, 73.23, -7.34) mm, rotated rx 180 ry 0 rz 90 deg; joints [76.392, -17.436, 84.182, 0, 23.254, 76.392]
  MoveL 5059 to (21.26, 73.4, -7.75) mm, rotated rx -180 ry 0 rz 90 deg; joints [76.386, -17.445, 84.28, 0, 23.164, 76.386]
  MoveC 5060 to (-2.01, 73.82, -7.75) mm, rotated rx -180 ry 0 rz 90 deg; joints [76.213, -17.868, 85.943, 0, 21.925, 76.213] to (-25.28, 74.15, -7.75) mm, rotated rx 180 ry 0 rz 90 deg; joints [76.033, -18.265, 87.574, 0, 20.691, 76.033]
  MoveC 5061 to (-27.81, 70.98, -7.75) mm, rotated rx 180 ry 0 rz 90 deg; joints [75.905, -18.294, 87.694, 0, 20.6, 75.905] to (-27.42, 66.95, -7.75) mm, rotated rx 180 ry 0 rz 90 deg; joints [75.773, -18.271, 87.597, 0, 20.674, 75.773]
  MoveL 5062 to (-9.35, 55.44, -7.75) mm, rotated rx 180 ry 0 rz 90 deg; joints [75.544, -17.916, 86.134, 0, 21.781, 75.544]
  MoveC 5063 to (-8.92, 55.2, -7.75) mm, rotated rx -180 ry 0 rz 90 deg; joints [75.54, -17.907, 86.099, 0, 21.808, 75.54] to (-8.45, 55.01, -7.75) mm, rotated rx -180 ry 0 rz 90 deg; joints [75.538, -17.898, 86.063, 0, 21.835, 75.538]
  MoveC 5064 to (-7.64, 54.93, -7.75) mm, rotated rx 180 ry 0 rz 90 deg; joints [75.542, -17.883, 86.004, 0, 21.879, 75.542] to (-6.81, 54.95, -7.75) mm, rotated rx 180 ry 0 rz 90 deg; joints [75.549, -17.869, 85.947, 0, 21.922, 75.549]
  MoveL 5065 to (-6.16, 55.01, -7.75) mm, rotated rx -180 ry 0 rz 90 deg; joints [75.557, -17.858, 85.902, 0, 21.956, 75.557]
  MoveC 5066 to (9.95, 56.19, -7.75) mm, rotated rx -180 ry 0 rz 90 deg; joints [75.731, -17.575, 84.783, 0, 22.791, 75.731] to (26.06, 57.44, -7.75) mm, rotated rx -180 ry 0 rz 90 deg; joints [75.905, -17.28, 83.651, 0, 23.629, 75.905]
  MoveC 5067 to (43.62, 59.08, -7.75) mm, rotated rx 180 ry 0 rz 90 deg; joints [76.099, -16.946, 82.404, 0, 24.542, 76.099] to (61.12, 61.19, -7.75) mm, rotated rx -180 ry 0 rz 90 deg; joints [76.304, -16.601, 81.151, 0, 25.45, 76.304]
  MoveL 5068 to (62.07, 61.33, -7.75) mm, rotated rx 180 ry 0 rz 90 deg; joints [76.316, -16.582, 81.083, 0, 25.499, 76.316]
  MoveL 5069 to (68.32, 62.31, -7.75) mm, rotated rx 180 ry 0 rz 90 deg; joints [76.396, -16.456, 80.635, 0, 25.822, 76.396]
  MoveC 5070 to (69.83, 63.12, -7.75) mm, rotated rx -180 ry 0 rz 90 deg; joints [76.433, -16.428, 80.535, 0, 25.893, 76.433] to (70.53, 64.69, -7.75) mm, rotated rx 180 ry 0 rz 90 deg; joints [76.488, -16.421, 80.511, 0, 25.91, 76.488]
  MoveL 5071 to (70.55, 64.91, -7.75) mm, rotated rx 180 ry 0 rz 90 deg; joints [76.496, -16.422, 80.514, 0, 25.908, 76.496]
  MoveL 5072 to (70.55, 68.7, -7.75) mm, rotated rx 180 ry 0 rz 90 deg; joints [76.616, -16.441, 80.582, 0, 25.859, 76.616]
  MoveL 5073 to (70.54, 68.92, -7.75) mm, rotated rx 180 ry 0 rz 90 deg; joints [76.623, -16.443, 80.587, 0, 25.856, 76.623]
  MoveC 5074 to (69.81, 70.55, -7.75) mm, rotated rx -180 ry 0 rz 90 deg; joints [76.669, -16.466, 80.671, 0, 25.796, 76.669] to (68.19, 71.29, -7.75) mm, rotated rx 180 ry 0 rz 90 deg; joints [76.681, -16.504, 80.805, 0, 25.699, 76.681]
  MoveC 5075 to (46.66, 72.59, -7.75) mm, rotated rx -180 ry 0 rz 90 deg; joints [76.558, -16.951, 82.422, 0, 24.529, 76.558] to (25.11, 73.32, -7.75) mm, rotated rx 180 ry 0 rz 90 deg; joints [76.414, -17.372, 84.001, 0, 23.37, 76.414]
  MoveC 5076 to (23.19, 73.36, -7.75) mm, rotated rx 180 ry 0 rz 90 deg; joints [76.4, -17.408, 84.141, 0, 23.267, 76.4] to (21.26, 73.4, -7.75) mm, rotated rx -180 ry 0 rz 90 deg; joints [76.386, -17.445, 84.28, 0, 23.164, 76.386]
  MoveL 5077 to (21.11, 65.85, -7.75) mm, rotated rx -180 ry 0 rz 90 deg; joints [76.138, -17.413, 84.158, 0, 23.255, 76.138]
  MoveL 5078 to (21.11, 65.85, -4.75) mm, rotated rx 180 ry 0 rz 90 deg; joints [76.138, -17.566, 84.26, 0, 23.306, 76.138]
  Establecer velocidad (1000.0 mm/s)
  MoveL 5079 to (21.11, 65.85, 10) mm, rotated rx -180 ry 0 rz 90 deg; joints [76.138, -18.319, 84.753, 0, 23.567, 76.138]
  Establecer velocidad (66.7 mm/s)
  MoveL 5080 to (36.11, 20.92, 10) mm, rotated rx -180 ry 0 rz 90 deg; joints [74.813, -17.798, 82.825, 0, 24.973, 74.813]
  MoveL 5081 to (36.11, 20.92, -4.5) mm, rotated rx -180 ry 0 rz 90 deg; joints [74.813, -17.063, 82.34, 0, 24.723, 74.813]
  MoveL 5082 to (36.26, 22.43, -4.91) mm, rotated rx 180 ry 0 rz 90 deg; joints [74.863, -17.048, 82.345, 0, 24.703, 74.863]
  MoveL 5083 to (36.05, 23.94, -5.31) mm, rotated rx -180 ry 0 rz 90 deg; joints [74.909, -17.039, 82.376, 0, 24.663, 74.909]
  MoveL 5084 to (35.51, 25.36, -5.72) mm, rotated rx 180 ry 0 rz 90 deg; joints [74.95, -17.037, 82.429, 0, 24.608, 74.95]
  MoveL 5085 to (34.67, 26.62, -6.12) mm, rotated rx -180 ry 0 rz 90 deg; joints [74.983, -17.04, 82.502, 0, 24.538, 74.983]
  MoveL 5086 to (33.57, 27.67, -6.53) mm, rotated rx 180 ry 0 rz 90 deg; joints [75.007, -17.046, 82.588, 0, 24.458, 75.007]
  MoveL 5087 to (32.27, 28.45, -6.94) mm, rotated rx 180 ry 0 rz 90 deg; joints [75.021, -17.056, 82.684, 0, 24.371, 75.021]
  MoveL 5088 to (30.82, 28.92, -7.34) mm, rotated rx -180 ry 0 rz 90 deg; joints [75.024, -17.066, 82.785, 0, 24.281, 75.024]
  MoveL 5089 to (29.31, 29.03, -7.75) mm, rotated rx 180 ry 0 rz 90 deg; joints [75.014, -17.075, 82.883, 0, 24.192, 75.014]
  MoveL 5090 to (10.9, 28.68, -7.75) mm, rotated rx 180 ry 0 rz 90 deg; joints [74.843, -17.424, 84.201, 0, 23.223, 74.843]
  MoveL 5091 to (9.95, 28.61, -7.75) mm, rotated rx 180 ry 0 rz 90 deg; joints [74.833, -17.441, 84.267, 0, 23.174, 74.833]
  MoveC 5092 to (7.54, 26.99, -7.75) mm, rotated rx -180 ry 0 rz 90 deg; joints [74.758, -17.478, 84.407, 0, 23.07, 74.758] to (6.82, 24.17, -7.75) mm, rotated rx 180 ry 0 rz 90 deg; joints [74.66, -17.477, 84.403, 0, 23.073, 74.66]
  MoveL 5093 to (6.95, 23.73, -7.75) mm, rotated rx -180 ry 0 rz 90 deg; joints [74.648, -17.472, 84.386, 0, 23.086, 74.648]
  MoveL 5094 to (11.63, 10.9, -7.75) mm, rotated rx 180 ry 0 rz 90 deg; joints [74.274, -17.318, 83.798, 0, 23.521, 74.274]
  MoveL 5095 to (12.05, 9.74, -7.75) mm, rotated rx 180 ry 0 rz 90 deg; joints [74.241, -17.304, 83.744, 0, 23.56, 74.241]
  MoveC 5096 to (12.56, 8.81, -7.75) mm, rotated rx -180 ry 0 rz 90 deg; joints [74.215, -17.29, 83.689, 0, 23.601, 74.215] to (13.3, 8.04, -7.75) mm, rotated rx 180 ry 0 rz 90 deg; joints [74.198, -17.271, 83.62, 0, 23.652, 74.198]
  MoveL 5097 to (27.96, -3.17, -7.75) mm, rotated rx -180 ry 0 rz 90 deg; joints [73.972, -16.926, 82.333, 0, 24.594, 73.972]
  MoveL 5098 to (28.9, -3.84, -7.75) mm, rotated rx 180 ry 0 rz 90 deg; joints [73.96, -16.904, 82.25, 0, 24.654, 73.96]
  MoveC 5099 to (31.69, -3.99, -7.75) mm, rotated rx 180 ry 0 rz 90 deg; joints [73.981, -16.848, 82.044, 0, 24.804, 73.981] to (33.98, -2.37, -7.75) mm, rotated rx -180 ry 0 rz 90 deg; joints [74.053, -16.811, 81.912, 0, 24.9, 74.053]
  MoveL 5100 to (51.41, 22.3, -7.75) mm, rotated rx 180 ry 0 rz 90 deg; joints [74.989, -16.596, 81.133, 0, 25.463, 74.989]
  MoveL 5101 to (51.65, 22.67, -7.75) mm, rotated rx 180 ry 0 rz 90 deg; joints [75.002, -16.593, 81.123, 0, 25.47, 75.002]
  MoveC 5102 to (51.27, 26.48, -7.75) mm, rotated rx 180 ry 0 rz 90 deg; joints [75.12, -16.622, 81.225, 0, 25.396, 75.12] to (48.67, 29.28, -7.75) mm, rotated rx -180 ry 0 rz 90 deg; joints [75.187, -16.69, 81.472, 0, 25.218, 75.187]
  MoveL 5103 to (48.33, 29.3, -7.75) mm, rotated rx 180 ry 0 rz 90 deg; joints [75.185, -16.697, 81.498, 0, 25.2, 75.185]
  MoveL 5104 to (34.59, 29.13, -7.75) mm, rotated rx 180 ry 0 rz 90 deg; joints [75.063, -16.972, 82.501, 0, 24.471, 75.063]
  MoveL 5105 to (29.31, 29.03, -7.75) mm, rotated rx 180 ry 0 rz 90 deg; joints [75.014, -17.075, 82.883, 0, 24.192, 75.014]
  MoveL 5106 to (29.45, 21.49, -7.75) mm, rotated rx 180 ry 0 rz 90 deg; joints [74.774, -17.033, 82.725, 0, 24.308, 74.774]
  MoveL 5107 to (29.45, 21.49, -4.75) mm, rotated rx 180 ry 0 rz 90 deg; joints [74.774, -17.185, 82.827, 0, 24.359, 74.774]
  Establecer velocidad (1000.0 mm/s)
  MoveL 5108 to (29.45, 21.49, 10) mm, rotated rx -180 ry 0 rz 90 deg; joints [74.774, -17.934, 83.32, 0, 24.614, 74.774]
  Establecer velocidad (66.7 mm/s)
  MoveL 5109 to (63.42, -31.65, 10) mm, rotated rx -180 ry 0 rz 90 deg; joints [73.404, -16.908, 79.7, 0, 27.207, 73.404]
  MoveL 5110 to (63.42, -31.65, -4.5) mm, rotated rx -180 ry 0 rz 90 deg; joints [73.404, -16.181, 79.212, 0, 26.969, 73.404]
  MoveL 5111 to (64.92, -31.83, -4.91) mm, rotated rx 180 ry 0 rz 90 deg; joints [73.412, -16.126, 79.081, 0, 27.045, 73.412]
  MoveL 5112 to (66.43, -31.65, -5.31) mm, rotated rx 180 ry 0 rz 90 deg; joints [73.432, -16.074, 78.958, 0, 27.116, 73.432]
  MoveL 5113 to (67.86, -31.14, -5.72) mm, rotated rx -180 ry 0 rz 90 deg; joints [73.461, -16.025, 78.847, 0, 27.178, 73.461]
  MoveL 5114 to (69.14, -30.32, -6.12) mm, rotated rx 180 ry 0 rz 90 deg; joints [73.498, -15.982, 78.755, 0, 27.227, 73.498]
  MoveL 5115 to (70.21, -29.24, -6.53) mm, rotated rx -180 ry 0 rz 90 deg; joints [73.541, -15.945, 78.685, 0, 27.261, 73.541]
  MoveL 5116 to (71.02, -27.96, -6.94) mm, rotated rx 180 ry 0 rz 90 deg; joints [73.588, -15.915, 78.639, 0, 27.277, 73.588]
  MoveL 5117 to (71.52, -26.52, -7.34) mm, rotated rx 180 ry 0 rz 90 deg; joints [73.637, -15.893, 78.619, 0, 27.274, 73.637]
  MoveL 5118 to (71.66, -25.01, -7.75) mm, rotated rx 180 ry 0 rz 90 deg; joints [73.685, -15.88, 78.628, 0, 27.252, 73.685]
  MoveL 5119 to (71.66, -15.3, -7.75) mm, rotated rx 180 ry 0 rz 90 deg; joints [73.986, -15.942, 78.841, 0, 27.101, 73.986]
  MoveC 5120 to (69.39, -12.27, -7.75) mm, rotated rx 180 ry 0 rz 90 deg; joints [74.06, -16.011, 79.077, 0, 26.933, 74.06] to (65.86, -10.89, -7.75) mm, rotated rx -180 ry 0 rz 90 deg; joints [74.071, -16.096, 79.372, 0, 26.724, 74.071]
  MoveL 5121 to (64.77, -11.03, -7.75) mm, rotated rx 180 ry 0 rz 90 deg; joints [74.057, -16.119, 79.451, 0, 26.668, 74.057]
  MoveL 5122 to (55.36, -23.84, -7.75) mm, rotated rx 180 ry 0 rz 90 deg; joints [73.573, -16.241, 79.877, 0, 26.364, 73.573]
  MoveC 5123 to (54.69, -26.04, -7.75) mm, rotated rx 180 ry 0 rz 90 deg; joints [73.498, -16.241, 79.878, 0, 26.364, 73.498] to (55.56, -28.17, -7.75) mm, rotated rx -180 ry 0 rz 90 deg; joints [73.439, -16.209, 79.766, 0, 26.444, 73.439]
  MoveL 5124 to (65.16, -38.93, -7.75) mm, rotated rx -180 ry 0 rz 90 deg; joints [73.195, -15.932, 78.806, 0, 27.126, 73.195]
  MoveC 5125 to (67.47, -38.77, -7.75) mm, rotated rx 180 ry 0 rz 90 deg; joints [73.221, -15.882, 78.635, 0, 27.247, 73.221] to (69.53, -37.7, -7.75) mm, rotated rx -180 ry 0 rz 90 deg; joints [73.273, -15.843, 78.504, 0, 27.339, 73.273]
  MoveC 5126 to (70.79, -36.35, -7.75) mm, rotated rx 180 ry 0 rz 90 deg; joints [73.327, -15.824, 78.439, 0, 27.385, 73.327] to (71.66, -34.72, -7.75) mm, rotated rx 180 ry 0 rz 90 deg; joints [73.385, -15.816, 78.411, 0, 27.405, 73.385]
  MoveL 5127 to (71.66, -25.01, -7.75) mm, rotated rx 180 ry 0 rz 90 deg; joints [73.685, -15.88, 78.628, 0, 27.252, 73.685]
  MoveL 5128 to (64.1, -25.01, -7.75) mm, rotated rx 180 ry 0 rz 90 deg; joints [73.616, -16.045, 79.197, 0, 26.849, 73.616]
  MoveL 5129 to (64.1, -25.01, -4.75) mm, rotated rx -180 ry 0 rz 90 deg; joints [73.616, -16.196, 79.299, 0, 26.897, 73.616]
  Establecer velocidad (1000.0 mm/s)
  MoveL 5130 to (64.1, -25.01, 10) mm, rotated rx 180 ry 0 rz 90 deg; joints [73.616, -16.936, 79.796, 0, 27.14, 73.616]
  Establecer velocidad (66.7 mm/s)
  MoveL 5131 to (16.49, -65.49, 10) mm, rotated rx 180 ry 0 rz 90 deg; joints [71.892, -17.673, 82.374, 0, 25.299, 71.892]
  MoveL 5132 to (16.49, -65.49, -4.5) mm, rotated rx -180 ry 0 rz 90 deg; joints [71.892, -16.939, 81.888, 0, 25.051, 71.892]
  MoveL 5133 to (16.33, -67, -4.91) mm, rotated rx 180 ry 0 rz 90 deg; joints [71.843, -16.912, 81.85, 0, 25.062, 71.843]
  MoveL 5134 to (16.55, -68.5, -5.31) mm, rotated rx -180 ry 0 rz 90 deg; joints [71.798, -16.877, 81.785, 0, 25.092, 71.798]
  MoveL 5135 to (17.08, -69.92, -5.72) mm, rotated rx -180 ry 0 rz 90 deg; joints [71.759, -16.837, 81.699, 0, 25.138, 71.759]
  MoveL 5136 to (17.92, -71.19, -6.12) mm, rotated rx -180 ry 0 rz 90 deg; joints [71.728, -16.791, 81.594, 0, 25.197, 71.728]
  MoveL 5137 to (19.02, -72.24, -6.53) mm, rotated rx -180 ry 0 rz 90 deg; joints [71.707, -16.741, 81.475, 0, 25.266, 71.707]
  MoveL 5138 to (20.33, -73.02, -6.94) mm, rotated rx 180 ry 0 rz 90 deg; joints [71.696, -16.689, 81.348, 0, 25.341, 71.696]
  MoveL 5139 to (21.78, -73.49, -7.34) mm, rotated rx 180 ry 0 rz 90 deg; joints [71.696, -16.636, 81.218, 0, 25.418, 71.696]
  MoveL 5140 to (23.29, -73.6, -7.75) mm, rotated rx 180 ry 0 rz 90 deg; joints [71.708, -16.584, 81.092, 0, 25.493, 71.708]
  MoveC 5141 to (35.3, -73.34, -7.75) mm, rotated rx -180 ry 0 rz 90 deg; joints [71.839, -16.339, 80.22, 0, 26.119, 71.839] to (47.3, -73.05, -7.75) mm, rotated rx 180 ry 0 rz 90 deg; joints [71.969, -16.087, 79.341, 0, 26.746, 71.969]
  MoveC 5142 to (49.88, -70.01, -7.75) mm, rotated rx -180 ry 0 rz 90 deg; joints [72.089, -16.053, 79.222, 0, 26.83, 72.089] to (50.02, -66.03, -7.75) mm, rotated rx -180 ry 0 rz 90 deg; joints [72.213, -16.077, 79.307, 0, 26.77, 72.213]
  MoveC 5143 to (37.62, -51.34, -7.75) mm, rotated rx 180 ry 0 rz 90 deg; joints [72.546, -16.438, 80.569, 0, 25.869, 72.546] to (25.11, -36.74, -7.75) mm, rotated rx -180 ry 0 rz 90 deg; joints [72.882, -16.785, 81.814, 0, 24.97, 72.882]
  MoveL 5144 to (24.83, -36.48, -7.75) mm, rotated rx -180 ry 0 rz 90 deg; joints [72.887, -16.792, 81.84, 0, 24.952, 72.887]
  MoveL 5145 to (12.32, -26.4, -7.75) mm, rotated rx -180 ry 0 rz 90 deg; joints [73.085, -17.097, 82.966, 0, 24.132, 73.085]
  MoveC 5146 to (9.12, -25.98, -7.75) mm, rotated rx 180 ry 0 rz 90 deg; joints [73.068, -17.161, 83.204, 0, 23.957, 73.068] to (6.57, -27.96, -7.75) mm, rotated rx 180 ry 0 rz 90 deg; joints [72.98, -17.198, 83.343, 0, 23.855, 72.98]
  MoveL 5147 to (6.29, -28.9, -7.75) mm, rotated rx 180 ry 0 rz 90 deg; joints [72.947, -17.198, 83.343, 0, 23.855, 72.947]
  MoveL 5148 to (-4.48, -69.16, -7.75) mm, rotated rx 180 ry 0 rz 90 deg; joints [71.558, -17.158, 83.192, 0, 23.966, 71.558]
  MoveC 5149 to (-3.8, -72.51, -7.75) mm, rotated rx 180 ry 0 rz 90 deg; joints [71.46, -17.124, 83.064, 0, 24.059, 71.46] to (-0.73, -73.99, -7.75) mm, rotated rx -180 ry 0 rz 90 deg; joints [71.446, -17.056, 82.81, 0, 24.245, 71.446]
  MoveC 5150 to (11.28, -73.81, -7.75) mm, rotated rx -180 ry 0 rz 90 deg; joints [71.577, -16.823, 81.955, 0, 24.868, 71.577] to (23.29, -73.6, -7.75) mm, rotated rx 180 ry 0 rz 90 deg; joints [71.708, -16.584, 81.092, 0, 25.493, 71.708]
  MoveL 5151 to (23.14, -66.05, -7.75) mm, rotated rx -180 ry 0 rz 90 deg; joints [71.942, -16.638, 81.283, 0, 25.355, 71.942]
  MoveL 5152 to (23.14, -66.05, -4.75) mm, rotated rx 180 ry 0 rz 90 deg; joints [71.942, -16.789, 81.385, 0, 25.405, 71.942]
  Establecer velocidad (1000.0 mm/s)
  MoveL 5153 to (23.14, -66.05, 10) mm, rotated rx 180 ry 0 rz 90 deg; joints [71.942, -17.534, 81.879, 0, 25.655, 71.942]
  Establecer velocidad (66.7 mm/s)
  MoveL 5154 to (-35.37, -51.31, 10) mm, rotated rx 180 ry 0 rz 90 deg; joints [71.802, -18.737, 86.362, 0, 22.375, 71.802]
  MoveL 5155 to (-35.37, -51.31, -4.5) mm, rotated rx -180 ry 0 rz 90 deg; joints [71.802, -17.991, 85.878, 0, 22.113, 71.802]
  MoveL 5156 to (-33.96, -51.87, -4.91) mm, rotated rx 180 ry 0 rz 90 deg; joints [71.799, -17.943, 85.754, 0, 22.189, 71.799]
  MoveL 5157 to (-32.45, -52.08, -5.31) mm, rotated rx 180 ry 0 rz 90 deg; joints [71.808, -17.895, 85.632, 0, 22.263, 71.808]
  MoveL 5158 to (-30.94, -51.94, -5.72) mm, rotated rx -180 ry 0 rz 90 deg; joints [71.829, -17.848, 85.516, 0, 22.332, 71.829]
  MoveL 5159 to (-29.49, -51.48, -6.12) mm, rotated rx -180 ry 0 rz 90 deg; joints [71.859, -17.804, 85.412, 0, 22.392, 71.859]
  MoveL 5160 to (-28.18, -50.7, -6.53) mm, rotated rx 180 ry 0 rz 90 deg; joints [71.898, -17.765, 85.325, 0, 22.44, 71.898]
  MoveL 5161 to (-27.08, -49.66, -6.94) mm, rotated rx -180 ry 0 rz 90 deg; joints [71.943, -17.731, 85.259, 0, 22.472, 71.943]
  MoveL 5162 to (-26.24, -48.39, -7.34) mm, rotated rx 180 ry 0 rz 90 deg; joints [71.993, -17.702, 85.215, 0, 22.487, 71.993]
  MoveL 5163 to (-25.72, -46.97, -7.75) mm, rotated rx 180 ry 0 rz 90 deg; joints [72.044, -17.68, 85.197, 0, 22.483, 72.044]
  MoveC 5164 to (-22.75, -35.57, -7.75) mm, rotated rx 180 ry 0 rz 90 deg; joints [72.442, -17.692, 85.245, 0, 22.448, 72.442] to (-19.79, -24.17, -7.75) mm, rotated rx 180 ry 0 rz 90 deg; joints [72.841, -17.703, 85.287, 0, 22.416, 72.841]
  MoveL 5165 to (-19.44, -22.74, -7.75) mm, rotated rx 180 ry 0 rz 90 deg; joints [72.891, -17.705, 85.293, 0, 22.411, 72.891]
  MoveL 5166 to (-19.43, -22.51, -7.75) mm, rotated rx 180 ry 0 rz 90 deg; joints [72.899, -17.706, 85.297, 0, 22.408, 72.899]
  MoveC 5167 to (-20.64, -19.94, -7.75) mm, rotated rx 180 ry 0 rz 90 deg; joints [72.97, -17.741, 85.437, 0, 22.304, 72.97] to (-23.22, -18.77, -7.75) mm, rotated rx -180 ry 0 rz 90 deg; joints [72.982, -17.793, 85.642, 0, 22.151, 72.982]
  MoveC 5168 to (-47.68, -23.92, -7.75) mm, rotated rx -180 ry 0 rz 90 deg; joints [72.566, -18.18, 87.219, 0, 20.962, 72.566] to (-72.13, -29.15, -7.75) mm, rotated rx 180 ry 0 rz 90 deg; joints [72.136, -18.542, 88.76, 0, 19.782, 72.136]
  MoveC 5169 to (-74.07, -30.34, -7.75) mm, rotated rx -180 ry 0 rz 90 deg; joints [72.076, -18.566, 88.865, 0, 19.702, 72.076] to (-74.83, -32.49, -7.75) mm, rotated rx 180 ry 0 rz 90 deg; joints [71.996, -18.567, 88.869, 0, 19.699, 71.996]
  MoveL 5170 to (-74.83, -70.6, -7.75) mm, rotated rx 180 ry 0 rz 90 deg; joints [70.739, -18.368, 88.008, 0, 20.36, 70.739]
  MoveC 5171 to (-73.92, -73.06, -7.75) mm, rotated rx 180 ry 0 rz 90 deg; joints [70.669, -18.34, 87.89, 0, 20.45, 70.669] to (-71.55, -74.17, -7.75) mm, rotated rx -180 ry 0 rz 90 deg; joints [70.66, -18.296, 87.704, 0, 20.592, 70.66]
  MoveL 5172 to (-70.6, -74.2, -7.75) mm, rotated rx -180 ry 0 rz 90 deg; joints [70.67, -18.281, 87.64, 0, 20.641, 70.67]
  MoveL 5173 to (-65.86, -74.16, -7.75) mm, rotated rx 180 ry 0 rz 90 deg; joints [70.725, -18.205, 87.321, 0, 20.884, 70.725]
  MoveL 5174 to (-63.97, -74.15, -7.75) mm, rotated rx 180 ry 0 rz 90 deg; joints [70.747, -18.174, 87.193, 0, 20.981, 70.747]
  MoveL 5175 to (-35.43, -73.91, -7.75) mm, rotated rx 180 ry 0 rz 90 deg; joints [71.074, -17.693, 85.247, 0, 22.446, 71.074]
  MoveC 5176 to (-33.36, -73.21, -7.75) mm, rotated rx 180 ry 0 rz 90 deg; joints [71.119, -17.661, 85.121, 0, 22.54, 71.119] to (-32.11, -71.41, -7.75) mm, rotated rx -180 ry 0 rz 90 deg; joints [71.19, -17.65, 85.077, 0, 22.573, 71.19]
  MoveL 5177 to (-31.88, -70.6, -7.75) mm, rotated rx 180 ry 0 rz 90 deg; joints [71.219, -17.65, 85.08, 0, 22.57, 71.219]
  MoveL 5178 to (-29.91, -63.02, -7.75) mm, rotated rx -180 ry 0 rz 90 deg; joints [71.483, -17.661, 85.121, 0, 22.54, 71.483]
  MoveL 5179 to (-29.42, -61.12, -7.75) mm, rotated rx -180 ry 0 rz 90 deg; joints [71.549, -17.663, 85.131, 0, 22.533, 71.549]
  MoveC 5180 to (-27.57, -54.05, -7.75) mm, rotated rx 180 ry 0 rz 90 deg; joints [71.797, -17.672, 85.165, 0, 22.507, 71.797] to (-25.72, -46.97, -7.75) mm, rotated rx 180 ry 0 rz 90 deg; joints [72.044, -17.68, 85.197, 0, 22.483, 72.044]
  MoveL 5181 to (-33.03, -45.06, -7.75) mm, rotated rx -180 ry 0 rz 90 deg; joints [72.029, -17.819, 85.747, 0, 22.072, 72.029]
  MoveL 5182 to (-33.03, -45.06, -4.75) mm, rotated rx 180 ry 0 rz 90 deg; joints [72.029, -17.973, 85.849, 0, 22.125, 72.029]
  Establecer velocidad (1000.0 mm/s)
  MoveL 5183 to (-33.03, -45.06, 10) mm, rotated rx 180 ry 0 rz 90 deg; joints [72.029, -18.731, 86.341, 0, 22.391, 72.029]
  Establecer velocidad (66.7 mm/s)
  MoveL 5184 to (-66.59, 36.24, 10) mm, rotated rx 180 ry 0 rz 90 deg; joints [74.387, -19.685, 90.302, 0, 19.383, 74.387]
  MoveL 5185 to (-66.59, 36.24, -4.5) mm, rotated rx -180 ry 0 rz 90 deg; joints [74.387, -18.926, 89.818, 0, 19.108, 74.387]
  MoveL 5186 to (-68.1, 36.42, -4.91) mm, rotated rx 180 ry 0 rz 90 deg; joints [74.379, -18.928, 89.909, 0, 19.019, 74.379]
  MoveL 5187 to (-69.61, 36.24, -5.31) mm, rotated rx 180 ry 0 rz 90 deg; joints [74.358, -18.929, 89.993, 0, 18.936, 74.358]
  MoveL 5188 to (-71.04, 35.73, -5.72) mm, rotated rx -180 ry 0 rz 90 deg; joints [74.327, -18.927, 90.066, 0, 18.861, 74.327]
  MoveL 5189 to (-72.32, 34.91, -6.12) mm, rotated rx -180 ry 0 rz 90 deg; joints [74.287, -18.921, 90.122, 0, 18.798, 74.287]
  MoveL 5190 to (-73.39, 33.84, -6.53) mm, rotated rx -180 ry 0 rz 90 deg; joints [74.24, -18.911, 90.16, 0, 18.751, 74.24]
  MoveL 5191 to (-74.19, 32.55, -6.94) mm, rotated rx 180 ry 0 rz 90 deg; joints [74.189, -18.896, 90.175, 0, 18.72, 74.189]
  MoveL 5192 to (-74.69, 31.11, -7.34) mm, rotated rx -180 ry 0 rz 90 deg; joints [74.135, -18.876, 90.168, 0, 18.708, 74.135]
  MoveL 5193 to (-74.83, 29.6, -7.75) mm, rotated rx -180 ry 0 rz 90 deg; joints [74.082, -18.85, 90.134, 0, 18.716, 74.082]
  MoveL 5194 to (-74.83, 0.93, -7.75) mm, rotated rx -180 ry 0 rz 90 deg; joints [73.113, -18.726, 89.571, 0, 19.155, 73.113]
  MoveC 5195 to (-73.5, -1.83, -7.75) mm, rotated rx 180 ry 0 rz 90 deg; joints [73.034, -18.693, 89.426, 0, 19.267, 73.034] to (-70.52, -2.51, -7.75) mm, rotated rx -180 ry 0 rz 90 deg; joints [73.042, -18.645, 89.212, 0, 19.433, 73.042]
  MoveC 5196 to (-45.91, 3.13, -7.75) mm, rotated rx 180 ry 0 rz 90 deg; joints [73.477, -18.286, 87.662, 0, 20.624, 73.477] to (-21.32, 8.8, -7.75) mm, rotated rx -180 ry 0 rz 90 deg; joints [73.901, -17.902, 86.08, 0, 21.822, 73.901]
  MoveC 5197 to (-18.94, 10.6, -7.75) mm, rotated rx -180 ry 0 rz 90 deg; joints [73.982, -17.87, 85.951, 0, 21.919, 73.982] to (-18.71, 13.56, -7.75) mm, rotated rx 180 ry 0 rz 90 deg; joints [74.081, -17.881, 85.994, 0, 21.887, 74.081]
  MoveL 5198 to (-25.39, 32.22, -7.75) mm, rotated rx 180 ry 0 rz 90 deg; joints [74.635, -18.084, 86.822, 0, 21.263, 74.635]
  MoveC 5199 to (-25.93, 33.19, -7.75) mm, rotated rx -180 ry 0 rz 90 deg; joints [74.662, -18.098, 86.877, 0, 21.221, 74.662] to (-26.73, 33.96, -7.75) mm, rotated rx 180 ry 0 rz 90 deg; joints [74.68, -18.115, 86.947, 0, 21.168, 74.68]
  MoveL 5200 to (-27.01, 34.15, -7.75) mm, rotated rx -180 ry 0 rz 90 deg; joints [74.684, -18.12, 86.97, 0, 21.15, 74.684]
  MoveL 5201 to (-69.36, 61.3, -7.75) mm, rotated rx 180 ry 0 rz 90 deg; joints [75.215, -18.897, 90.351, 0, 18.547, 75.215]
  MoveC 5202 to (-69.96, 61.6, -7.75) mm, rotated rx -180 ry 0 rz 90 deg; joints [75.219, -18.907, 90.396, 0, 18.511, 75.219] to (-70.6, 61.77, -7.75) mm, rotated rx -180 ry 0 rz 90 deg; joints [75.219, -18.917, 90.442, 0, 18.475, 75.219]
  MoveC 5203 to (-73.09, 61.19, -7.75) mm, rotated rx -180 ry 0 rz 90 deg; joints [75.177, -18.951, 90.598, 0, 18.353, 75.177] to (-74.72, 59.23, -7.75) mm, rotated rx 180 ry 0 rz 90 deg; joints [75.095, -18.967, 90.672, 0, 18.294, 75.095]
  MoveC 5204 to (-74.8, 58.75, -7.75) mm, rotated rx -180 ry 0 rz 90 deg; joints [75.078, -18.966, 90.669, 0, 18.297, 75.078] to (-74.83, 58.27, -7.75) mm, rotated rx 180 ry 0 rz 90 deg; joints [75.061, -18.965, 90.663, 0, 18.302, 75.061]
  MoveL 5205 to (-74.83, 29.6, -7.75) mm, rotated rx -180 ry 0 rz 90 deg; joints [74.082, -18.85, 90.134, 0, 18.716, 74.082]
  MoveL 5206 to (-67.28, 29.6, -7.75) mm, rotated rx -180 ry 0 rz 90 deg; joints [74.155, -18.739, 89.629, 0, 19.11, 74.155]
  MoveL 5207 to (-67.28, 29.6, -4.75) mm, rotated rx 180 ry 0 rz 90 deg; joints [74.155, -18.896, 89.731, 0, 19.165, 74.155]
  Establecer velocidad (1000.0 mm/s)
  MoveL 5208 to (-67.28, 29.6, 10) mm, rotated rx 180 ry 0 rz 90 deg; joints [74.155, -19.667, 90.223, 0, 19.444, 74.155]
  Establecer velocidad (66.7 mm/s)
  MoveL 5209 to (-66.42, 36.24, 10) mm, rotated rx 180 ry 0 rz 90 deg; joints [74.388, -19.683, 90.291, 0, 19.392, 74.388]
  MoveL 5210 to (-66.42, 36.24, -4.75) mm, rotated rx 180 ry 0 rz 90 deg; joints [74.388, -18.911, 89.798, 0, 19.113, 74.388]
  MoveL 5211 to (-67.92, 36.42, -5.16) mm, rotated rx -180 ry 0 rz 90 deg; joints [74.38, -18.913, 89.889, 0, 19.024, 74.38]
  MoveL 5212 to (-69.43, 36.24, -5.56) mm, rotated rx 180 ry 0 rz 90 deg; joints [74.36, -18.913, 89.973, 0, 18.94, 74.36]
  MoveL 5213 to (-70.86, 35.73, -5.97) mm, rotated rx 180 ry 0 rz 90 deg; joints [74.329, -18.911, 90.046, 0, 18.865, 74.329]
  MoveL 5214 to (-72.15, 34.91, -6.38) mm, rotated rx -180 ry 0 rz 90 deg; joints [74.289, -18.905, 90.102, 0, 18.803, 74.289]
  MoveL 5215 to (-73.22, 33.84, -6.78) mm, rotated rx -180 ry 0 rz 90 deg; joints [74.242, -18.895, 90.14, 0, 18.755, 74.242]
  MoveL 5216 to (-74.02, 32.55, -7.19) mm, rotated rx 180 ry 0 rz 90 deg; joints [74.19, -18.88, 90.155, 0, 18.725, 74.19]
  MoveL 5217 to (-74.52, 31.11, -7.59) mm, rotated rx -180 ry 0 rz 90 deg; joints [74.137, -18.86, 90.148, 0, 18.712, 74.137]
  MoveL 5218 to (-74.66, 29.6, -8) mm, rotated rx 180 ry 0 rz 90 deg; joints [74.084, -18.835, 90.114, 0, 18.72, 74.084]
  MoveL 5219 to (-74.66, 1.42, -8) mm, rotated rx -180 ry 0 rz 90 deg; joints [73.132, -18.712, 89.561, 0, 19.151, 73.132]
  MoveL 5220 to (-74.62, 0.47, -8) mm, rotated rx -180 ry 0 rz 90 deg; joints [73.1, -18.707, 89.539, 0, 19.168, 73.1]
  MoveC 5221 to (-73.38, -1.63, -8) mm, rotated rx 180 ry 0 rz 90 deg; joints [73.042, -18.679, 89.413, 0, 19.266, 73.042] to (-71.07, -2.42, -8) mm, rotated rx -180 ry 0 rz 90 deg; joints [73.039, -18.641, 89.243, 0, 19.398, 73.039]
  MoveC 5222 to (-70.36, -2.31, -8) mm, rotated rx -180 ry 0 rz 90 deg; joints [73.05, -18.631, 89.197, 0, 19.433, 73.05] to (-69.65, -2.16, -8) mm, rotated rx 180 ry 0 rz 90 deg; joints [73.062, -18.621, 89.153, 0, 19.468, 73.062]
  MoveL 5223 to (-68.7, -1.92, -8) mm, rotated rx 180 ry 0 rz 90 deg; joints [73.08, -18.607, 89.094, 0, 19.513, 73.08]
  MoveC 5224 to (-45.01, 3.5, -8) mm, rotated rx -180 ry 0 rz 90 deg; joints [73.498, -18.26, 87.599, 0, 20.661, 73.498] to (-21.32, 8.98, -8) mm, rotated rx -180 ry 0 rz 90 deg; joints [73.907, -17.89, 86.076, 0, 21.815, 73.907]
  MoveC 5225 to (-19.09, 10.84, -8) mm, rotated rx 180 ry 0 rz 90 deg; joints [73.989, -17.861, 85.957, 0, 21.904, 73.989] to (-18.95, 13.74, -8) mm, rotated rx -180 ry 0 rz 90 deg; joints [74.085, -17.873, 86.006, 0, 21.867, 74.085]
  MoveL 5226 to (-25.53, 32.12, -8) mm, rotated rx 180 ry 0 rz 90 deg; joints [74.63, -18.073, 86.821, 0, 21.253, 74.63]
  MoveC 5227 to (-26.09, 33.13, -8) mm, rotated rx -180 ry 0 rz 90 deg; joints [74.658, -18.087, 86.879, 0, 21.208, 74.658] to (-26.95, 33.91, -8) mm, rotated rx 180 ry 0 rz 90 deg; joints [74.676, -18.105, 86.953, 0, 21.152, 74.676]
  MoveL 5228 to (-29.85, 35.78, -8) mm, rotated rx 180 ry 0 rz 90 deg; joints [74.712, -18.162, 87.189, 0, 20.973, 74.712]
  MoveL 5229 to (-69.18, 60.99, -8) mm, rotated rx -180 ry 0 rz 90 deg; joints [75.206, -18.88, 90.325, 0, 18.556, 75.206]
  MoveC 5230 to (-69.64, 61.25, -8) mm, rotated rx 180 ry 0 rz 90 deg; joints [75.21, -18.888, 90.36, 0, 18.528, 75.21] to (-70.13, 61.46, -8) mm, rotated rx 180 ry 0 rz 90 deg; joints [75.213, -18.896, 90.396, 0, 18.5, 75.213]
  MoveC 5231 to (-72.9, 60.98, -8) mm, rotated rx -180 ry 0 rz 90 deg; joints [75.172, -18.934, 90.573, 0, 18.361, 75.172] to (-74.63, 58.76, -8) mm, rotated rx 180 ry 0 rz 90 deg; joints [75.08, -18.95, 90.649, 0, 18.301, 75.08]
  MoveL 5232 to (-74.66, 57.33, -8) mm, rotated rx -180 ry 0 rz 90 deg; joints [75.031, -18.945, 90.626, 0, 18.32, 75.031]
  MoveL 5233 to (-74.66, 29.6, -8) mm, rotated rx 180 ry 0 rz 90 deg; joints [74.084, -18.835, 90.114, 0, 18.72, 74.084]
  MoveL 5234 to (-67.11, 29.6, -8) mm, rotated rx 180 ry 0 rz 90 deg; joints [74.157, -18.723, 89.609, 0, 19.114, 74.157]
  MoveL 5235 to (-67.11, 29.6, -5) mm, rotated rx 180 ry 0 rz 90 deg; joints [74.157, -18.88, 89.711, 0, 19.169, 74.157]
  Establecer velocidad (1000.0 mm/s)
  MoveL 5236 to (-67.11, 29.6, 10) mm, rotated rx 180 ry 0 rz 90 deg; joints [74.157, -19.665, 90.212, 0, 19.453, 74.157]
  Establecer velocidad (66.7 mm/s)
  MoveL 5237 to (-39.57, -30.81, 10) mm, rotated rx 180 ry 0 rz 90 deg; joints [72.424, -18.925, 87.107, 0, 21.817, 72.424]
  MoveL 5238 to (-39.57, -30.81, -4.75) mm, rotated rx -180 ry 0 rz 90 deg; joints [72.424, -18.164, 86.615, 0, 21.549, 72.424]
  MoveL 5239 to (-39.7, -29.3, -5.16) mm, rotated rx -180 ry 0 rz 90 deg; joints [72.472, -18.153, 86.643, 0, 21.51, 72.472]
  MoveL 5240 to (-40.2, -27.86, -5.56) mm, rotated rx -180 ry 0 rz 90 deg; joints [72.514, -18.148, 86.695, 0, 21.454, 72.514]
  MoveL 5241 to (-40.99, -26.57, -5.97) mm, rotated rx -180 ry 0 rz 90 deg; joints [72.548, -18.148, 86.764, 0, 21.384, 72.548]
  MoveL 5242 to (-42.06, -25.48, -6.38) mm, rotated rx 180 ry 0 rz 90 deg; joints [72.573, -18.15, 86.846, 0, 21.304, 72.573]
  MoveL 5243 to (-43.33, -24.66, -6.78) mm, rotated rx 180 ry 0 rz 90 deg; joints [72.586, -18.155, 86.938, 0, 21.217, 72.586]
  MoveL 5244 to (-44.76, -24.14, -7.19) mm, rotated rx -180 ry 0 rz 90 deg; joints [72.589, -18.16, 87.033, 0, 21.127, 72.589]
  MoveL 5245 to (-46.27, -23.95, -7.59) mm, rotated rx -180 ry 0 rz 90 deg; joints [72.58, -18.165, 87.127, 0, 21.038, 72.58]
  MoveL 5246 to (-47.78, -24.13, -8) mm, rotated rx 180 ry 0 rz 90 deg; joints [72.558, -18.168, 87.212, 0, 20.956, 72.558]
  MoveL 5247 to (-69.65, -28.78, -8) mm, rotated rx -180 ry 0 rz 90 deg; joints [72.175, -18.493, 88.593, 0, 19.899, 72.175]
  MoveL 5248 to (-71.83, -29.24, -8) mm, rotated rx 180 ry 0 rz 90 deg; joints [72.136, -18.524, 88.73, 0, 19.794, 72.136]
  MoveC 5249 to (-72.41, -29.4, -8) mm, rotated rx -180 ry 0 rz 90 deg; joints [72.125, -18.532, 88.765, 0, 19.768, 72.125] to (-72.95, -29.65, -8) mm, rotated rx 180 ry 0 rz 90 deg; joints [72.111, -18.539, 88.796, 0, 19.744, 72.111]
